KUKA KRL program: EPS_2_25716_MHCR06_A_20250905053017.src

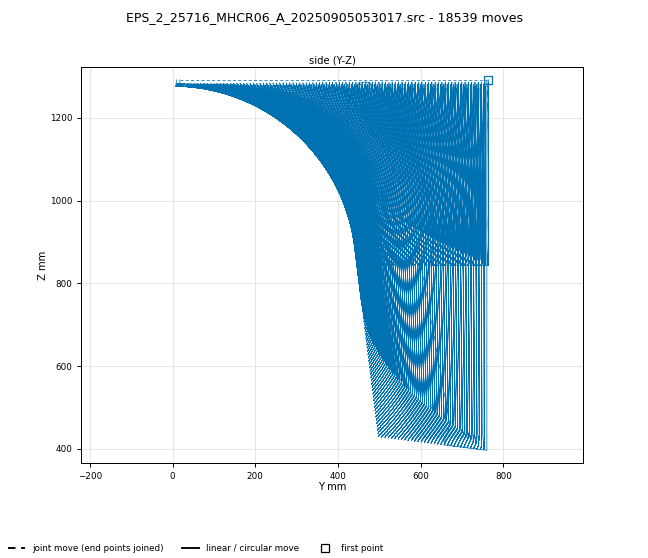
[picture p0: tool path of EPS_2_25716_MHCR06_A_20250905053017.src, 18539 of 18541 moves have a stored position in this frame; points joined in program order, loops and branches not executed]
&ACCESS RVP
&REL 4
&COMMENT QRS 19112012
&PARAM EDITMASK = *
DEF PART()
EXT BAS (BAS_COMMAND :IN,REAL :IN )
INT I
BAS (#INITMOV,0 )

;KUKA QRS Post kuka4.cps  Date:22-06-2017 !

File_ID=2806

QRS_PRE_INIT()

;Init var - Until changes are made in qrs_pre_init
Outlet_Square_prg=0
Inlet_1_Square_prg=0
Inlet_2_Square_prg=0
Inlet_3_Square_prg=0
Inlet_4_Square_prg=0
Inlet_5_Square_prg=0

Outlet_1={X 0.000, Y 457.000, Z 863.000, B 0.000, E1 0.000 }
Inlet_1={X 0.000, Y 457.000, Z 853.000, B 0.000, E1 180.000 }
Outlet_1_type=838
Inlet_1_type=838
;QRS#1=Sidecore dimensions
;QRS#2=825-33" Concrete
;QRS#3=825-33" Concrete
;QRS#4=
;QRS#5=
;QRS#6=
;QRS#7=
;QRS#8=
;QRS#9=S306-46
;QRS#10=S306-46
;QRS#11=
;QRS#12=
;QRS#13=
;QRS#14=
;QRS#15=
;QRS#16=1524x152x1753 5,75'
;QRS#17=EPS Height
;QRS#18=1282
;QRS#19=*
;QRS#20= UPDATED VERSION 22-06-2017
;QRS#21=*
Outlet_Square=0650
Inlet_1_Square=0650
Inlet_2_Square=0
Inlet_3_Square=0
Inlet_4_Square=0
Inlet_5_Square=0
Mill_Square=1
Outlet_Square_Prg=267
Inlet_1_Square_prg=267

QRS_INIT()

$ADVANCE=5

; T1
PTP {E1 176.612,E2 176.612}
PTP {X 0,Y 763.425,A -85,B 0,C 180,E1 176.612,E2 176.612,E3 0,E4 0,E5 0,E6 0}
QRS_SPEED_INIT()
LIN {X 0,Y 763.425,Z 1292,A -85,B 0,C 180,E1 176.612,E2 176.612,E3 0,E4 0,E5 0,E6 0} C_VEL
LIN {X 0,Y 763.425,Z 846.06,A -85,B 0,C 180,E1 176.612,E2 176.612} C_VEL
LIN {X 0,Y 763.534,Z 844.06,A -85,B 0,C 180,E1 176.762,E2 176.762} C_VEL
LIN {X 0,Y 763.871,Z 844.06,A -85,B 0,C 180,E1 177.187,E2 177.187} C_VEL
LIN {X 0,Y 763.823,Z 844.06,A -85,B 0,C 180,E1 184.692,E2 184.692} C_VEL
LIN {X 0,Y 763.818,Z 844.06,A -85,B 0,C 180,E1 192.28,E2 192.28} C_VEL
LIN {X 0,Y 763.836,Z 844.06,A -85,B 0,C 180,E1 200.095,E2 200.095} C_VEL
LIN {X 0,Y 763.785,Z 844.06,A -85,B 0,C 180,E1 208.327,E2 208.327} C_VEL
LIN {X 0,Y 762.377,Z 844.06,A -85,B 0,C 180,E1 210.541,E2 210.541} C_VEL
LIN {X 0,Y 762.698,Z 844.06,A -85,B 0,C 180,E1 214.994,E2 214.994} C_VEL
LIN {X 0,Y 763.696,Z 844.06,A -85,B 0,C 180,E1 216.695,E2 216.695} C_VEL
LIN {X 0,Y 763.424,Z 844.06,A -85,B 0,C 180,E1 224.741,E2 224.741} C_VEL
LIN {X 0,Y 763.668,Z 844.06,A -85,B 0,C 180,E1 225.277,E2 225.277} C_VEL
LIN {X 0,Y 763.811,Z 844.06,A -85,B 0,C 180,E1 233.406,E2 233.406} C_VEL
LIN {X 0,Y 763.414,Z 844.06,A -85,B 0,C 180,E1 233.624,E2 233.624} C_VEL
LIN {X 0,Y 763.044,Z 844.06,A -85,B 0,C 180,E1 233.668,E2 233.668} C_VEL
LIN {X 0,Y 762.773,Z 846.033,A -85,B 0,C 180,E1 233.717,E2 233.717} C_VEL
LIN {X 0,Y 763.464,Z 884.803,A -85,B 0,C 180,E1 234.197,E2 234.197} C_VEL
LIN {X 0,Y 763.74,Z 906.668,A -85,B 0,C 180,E1 234.483,E2 234.483} C_VEL
LIN {X 0,Y 763.751,Z 923.257,A -85,B 0,C 180,E1 234.748,E2 234.748} C_VEL
LIN {X 0,Y 763.617,Z 939.256,A -85,B 0,C 180,E1 235.054,E2 235.054} C_VEL
LIN {X 0,Y 763.249,Z 953.724,A -85,B 0,C 180,E1 235.362,E2 235.362} C_VEL
LIN {X 0,Y 763.625,Z 971.393,A -85,B 0,C 180,E1 235.846,E2 235.846} C_VEL
LIN {X 0,Y 763.699,Z 993.904,A -85,B 0,C 180,E1 236.542,E2 236.542} C_VEL
LIN {X 0,Y 763.605,Z 1014.167,A -85,B 0,C 180,E1 237.262,E2 237.262} C_VEL
LIN {X 0,Y 763.443,Z 1025.893,A -85,B 0,C 180,E1 237.721,E2 237.721} C_VEL
LIN {X 0,Y 763.576,Z 1034.178,A -85,B 0,C 180,E1 238.073,E2 238.073} C_VEL
LIN {X 0,Y 763.564,Z 1050.299,A -85,B 0,C 180,E1 238.794,E2 238.794} C_VEL
LIN {X 0,Y 763.558,Z 1067.921,A -85,B 0,C 180,E1 239.665,E2 239.665} C_VEL
LIN {X 0,Y 763.648,Z 1085.413,A -85,B 0,C 180,E1 240.62,E2 240.62} C_VEL
LIN {X 0,Y 763.58,Z 1101.247,A -85,B 0,C 180,E1 241.554,E2 241.554} C_VEL
LIN {X 0,Y 763.331,Z 1117.353,A -85,B 0,C 180,E1 242.582,E2 242.582} C_VEL
LIN {X 0,Y 763.287,Z 1132.396,A -85,B 0,C 180,E1 243.633,E2 243.633} C_VEL
LIN {X 0,Y 763.586,Z 1147.922,A -85,B 0,C 180,E1 244.824,E2 244.824} C_VEL
LIN {X 0,Y 763.68,Z 1158.714,A -85,B 0,C 180,E1 245.705,E2 245.705} C_VEL
LIN {X 0,Y 763.241,Z 1173.502,A -85,B 0,C 180,E1 246.987,E2 246.987} C_VEL
LIN {X 0,Y 763.107,Z 1186.863,A -85,B 0,C 180,E1 248.263,E2 248.263} C_VEL
LIN {X 0,Y 763.439,Z 1198.638,A -85,B 0,C 180,E1 249.493,E2 249.493} C_VEL
LIN {X 0,Y 763.75,Z 1205.883,A -85,B 0,C 180,E1 250.316,E2 250.316} C_VEL
LIN {X 0,Y 763.554,Z 1210.764,A -85,B 0,C 180,E1 250.869,E2 250.869} C_VEL
LIN {X 0,Y 762.975,Z 1220.993,A -85,B 0,C 180,E1 252.113,E2 252.113} C_VEL
LIN {X 0,Y 762.874,Z 1231.824,A -85,B 0,C 180,E1 253.584,E2 253.584} C_VEL
LIN {X 0,Y 763.518,Z 1241.781,A -85,B 0,C 180,E1 255.105,E2 255.105} C_VEL
LIN {X 0,Y 763.855,Z 1245.871,A -85,B 0,C 180,E1 255.793,E2 255.793} C_VEL
LIN {X 0,Y 763.464,Z 1249.702,A -85,B 0,C 180,E1 256.43,E2 256.43} C_VEL
LIN {X 0,Y 762.698,Z 1257.74,A -85,B 0,C 180,E1 257.94,E2 257.94} C_VEL
LIN {X 0,Y 762.694,Z 1264.404,A -85,B 0,C 180,E1 259.376,E2 259.376} C_VEL
LIN {X 0,Y 763.587,Z 1270.959,A -85,B 0,C 180,E1 261.054,E2 261.054} C_VEL
LIN {X 0,Y 763.866,Z 1272.551,A -85,B 0,C 180,E1 261.531,E2 261.531} C_VEL
LIN {X 0,Y 763.257,Z 1275.707,A -85,B 0,C 180,E1 262.472,E2 262.472} C_VEL
LIN {X 0,Y 762.641,Z 1279.586,A -85,B 0,C 180,E1 263.884,E2 263.884} C_VEL
LIN {X 0,Y 762.788,Z 1282.608,A -85,B 0,C 180,E1 265.299,E2 265.299} C_VEL
LIN {X 0,Y 763.582,Z 1284.794,A -85,B 0,C 180,E1 266.707,E2 266.707} C_VEL
LIN {X 0,Y 763.885,Z 1285.327,A -85,B 0,C 180,E1 267.185,E2 267.185} C_VEL
LIN {X 0,Y 762.666,Z 1286.718,A -85,B 0,C 180,E1 269.059,E2 269.059} C_VEL
LIN {X 0,Y 762.487,Z 1286.723,A -85,B 0,C 180,E1 270.937,E2 270.937} C_VEL
LIN {X 0,Y 763.544,Z 1285.349,A -85,B 0,C 180,E1 272.812,E2 272.812} C_VEL
LIN {X 0,Y 763.669,Z 1284.386,A -85,B 0,C 180,E1 273.591,E2 273.591} C_VEL
LIN {X 0,Y 763.006,Z 1282.612,A -85,B 0,C 180,E1 274.695,E2 274.695} C_VEL
LIN {X 0,Y 762.597,Z 1279.596,A -85,B 0,C 180,E1 276.112,E2 276.112} C_VEL
LIN {X 0,Y 762.981,Z 1275.722,A -85,B 0,C 180,E1 277.527,E2 277.527} C_VEL
LIN {X 0,Y 763.831,Z 1270.969,A -85,B 0,C 180,E1 278.939,E2 278.939} C_VEL
LIN {X 0,Y 763.296,Z 1267.291,A -85,B 0,C 180,E1 279.896,E2 279.896} C_VEL
LIN {X 0,Y 762.816,Z 1263.345,A -85,B 0,C 180,E1 280.857,E2 280.857} C_VEL
LIN {X 0,Y 762.703,Z 1256.562,A -85,B 0,C 180,E1 282.296,E2 282.296} C_VEL
LIN {X 0,Y 763.232,Z 1249.725,A -85,B 0,C 180,E1 283.57,E2 283.57} C_VEL
LIN {X 0,Y 763.817,Z 1243.189,A -85,B 0,C 180,E1 284.654,E2 284.654} C_VEL
LIN {X 0,Y 763.572,Z 1240.469,A -85,B 0,C 180,E1 285.11,E2 285.11} C_VEL
LIN {X 0,Y 762.935,Z 1230.124,A -85,B 0,C 180,E1 286.655,E2 286.655} C_VEL
LIN {X 0,Y 762.935,Z 1221.027,A -85,B 0,C 180,E1 287.883,E2 287.883} C_VEL
LIN {X 0,Y 763.482,Z 1209.87,A -85,B 0,C 180,E1 289.243,E2 289.243} C_VEL
LIN {X 0,Y 763.749,Z 1204.145,A -85,B 0,C 180,E1 289.879,E2 289.879} C_VEL
LIN {X 0,Y 763.45,Z 1196.64,A -85,B 0,C 180,E1 290.718,E2 290.718} C_VEL
LIN {X 0,Y 763.048,Z 1184.242,A -85,B 0,C 180,E1 291.997,E2 291.997} C_VEL
LIN {X 0,Y 763.138,Z 1172.143,A -85,B 0,C 180,E1 293.139,E2 293.139} C_VEL
LIN {X 0,Y 763.585,Z 1158.001,A -85,B 0,C 180,E1 294.356,E2 294.356} C_VEL
LIN {X 0,Y 763.639,Z 1146.811,A -85,B 0,C 180,E1 295.265,E2 295.265} C_VEL
LIN {X 0,Y 763.318,Z 1130.65,A -85,B 0,C 180,E1 296.492,E2 296.492} C_VEL
LIN {X 0,Y 763.302,Z 1114.416,A -85,B 0,C 180,E1 297.612,E2 297.612} C_VEL
LIN {X 0,Y 763.543,Z 1098.417,A -85,B 0,C 180,E1 298.618,E2 298.618} C_VEL
LIN {X 0,Y 763.622,Z 1082.558,A -85,B 0,C 180,E1 299.543,E2 299.543} C_VEL
LIN {X 0,Y 763.573,Z 1064.988,A -85,B 0,C 180,E1 300.484,E2 300.484} C_VEL
LIN {X 0,Y 763.534,Z 1047.236,A -85,B 0,C 180,E1 301.35,E2 301.35} C_VEL
LIN {X 0,Y 763.593,Z 1029.838,A -85,B 0,C 180,E1 302.115,E2 302.115} C_VEL
LIN {X 0,Y 763.413,Z 1015.501,A -85,B 0,C 180,E1 302.694,E2 302.694} C_VEL
LIN {X 0,Y 763.608,Z 1006.295,A -85,B 0,C 180,E1 303.025,E2 303.025} C_VEL
LIN {X 0,Y 763.703,Z 991.031,A -85,B 0,C 180,E1 303.552,E2 303.552} C_VEL
LIN {X 0,Y 763.676,Z 970.59,A -85,B 0,C 180,E1 304.173,E2 304.173} C_VEL
LIN {X 0,Y 763.496,Z 952.918,A -85,B 0,C 180,E1 304.645,E2 304.645} C_VEL
LIN {X 0,Y 763.248,Z 942.803,A -85,B 0,C 180,E1 304.891,E2 304.891} C_VEL
LIN {X 0,Y 763.633,Z 926.104,A -85,B 0,C 180,E1 305.206,E2 305.206} C_VEL
LIN {X 0,Y 763.708,Z 908.879,A -85,B 0,C 180,E1 305.487,E2 305.487} C_VEL
LIN {X 0,Y 763.624,Z 893.145,A -85,B 0,C 180,E1 305.699,E2 305.699} C_VEL
LIN {X 0,Y 762.84,Z 848.075,A -85,B 0,C 180,E1 306.256,E2 306.256} C_VEL
LIN {X 0,Y 763.386,Z 844.06,A -85,B 0,C 180,E1 306.373,E2 306.373} C_VEL
LIN {X 0,Y 763.822,Z 844.06,A -85,B 0,C 180,E1 306.471,E2 306.471} C_VEL
LIN {X 0,Y 763.69,Z 844.06,A -85,B 0,C 180,E1 312.133,E2 312.133} C_VEL
LIN {X 0,Y 763.519,Z 844.06,A -85,B 0,C 180,E1 312.562,E2 312.562} C_VEL
LIN {X 0,Y 763.784,Z 844.06,A -85,B 0,C 180,E1 320.259,E2 320.259} C_VEL
LIN {X 0,Y 763.636,Z 844.06,A -85,B 0,C 180,E1 326.569,E2 326.569} C_VEL
LIN {X 0,Y 763.395,Z 844.06,A -85,B 0,C 180,E1 327.301,E2 327.301} C_VEL
LIN {X 0,Y 763.767,Z 844.06,A -85,B 0,C 180,E1 333.782,E2 333.782} C_VEL
LIN {X 0,Y 763.774,Z 844.06,A -85,B 0,C 180,E1 341.888,E2 341.888} C_VEL
LIN {X 0,Y 763.762,Z 844.06,A -85,B 0,C 180,E1 349.631,E2 349.631} C_VEL
LIN {X 0,Y 763.87,Z 844.06,A -85,B 0,C 180,E1 357.187,E2 357.187} C_VEL
LIN {X 0,Y 763.811,Z 844.06,A -85,B 0,C 180,E1 364.692,E2 364.692} C_VEL
LIN {X 0,Y 763.783,Z 844.06,A -85,B 0,C 180,E1 372.281,E2 372.281} C_VEL
LIN {X 0,Y 763.826,Z 844.06,A -85,B 0,C 180,E1 380.095,E2 380.095} C_VEL
LIN {X 0,Y 763.817,Z 844.06,A -85,B 0,C 180,E1 388.325,E2 388.325} C_VEL
LIN {X 0,Y 762.037,Z 844.06,A -85,B 0,C 180,E1 393.248,E2 393.248} C_VEL
LIN {X 0,Y 762.694,Z 844.06,A -85,B 0,C 180,E1 394.994,E2 394.994} C_VEL
LIN {X 0,Y 763.695,Z 844.06,A -85,B 0,C 180,E1 396.702,E2 396.702} C_VEL
LIN {X 0,Y 763.462,Z 844.06,A -85,B 0,C 180,E1 404.738,E2 404.738} C_VEL
LIN {X 0,Y 763.718,Z 844.06,A -85,B 0,C 180,E1 405.287,E2 405.287} C_VEL
LIN {X 0,Y 763.716,Z 844.06,A -85,B 0,C 180,E1 413.316,E2 413.316} C_VEL
LIN {X 0,Y 763.638,Z 844.06,A -85,B 0,C 180,E1 413.584,E2 413.584} C_VEL
LIN {X 0,Y 762.291,Z 846.452,A -85,B 0,C 180,E1 413.765,E2 413.765} C_VEL
LIN {X 0,Y 763.273,Z 877.101,A -85,B 0,C 180,E1 414.168,E2 414.168} C_VEL
LIN {X 0,Y 763.588,Z 897.131,A -85,B 0,C 180,E1 414.436,E2 414.436} C_VEL
LIN {X 0,Y 763.619,Z 912.565,A -85,B 0,C 180,E1 414.683,E2 414.683} C_VEL
LIN {X 0,Y 763.39,Z 929.413,A -85,B 0,C 180,E1 415,E2 415} C_VEL
LIN {X 0,Y 763.232,Z 936.778,A -85,B 0,C 180,E1 415.154,E2 415.154} C_VEL
LIN {X 0,Y 763.582,Z 953.603,A -85,B 0,C 180,E1 415.585,E2 415.585} C_VEL
LIN {X 0,Y 763.631,Z 965.787,A -85,B 0,C 180,E1 415.931,E2 415.931} C_VEL
LIN {X 0,Y 763.567,Z 984.677,A -85,B 0,C 180,E1 416.518,E2 416.518} C_VEL
LIN {X 0,Y 763.383,Z 997.385,A -85,B 0,C 180,E1 416.957,E2 416.957} C_VEL
LIN {X 0,Y 763.555,Z 1005.386,A -85,B 0,C 180,E1 417.264,E2 417.264} C_VEL
LIN {X 0,Y 763.596,Z 1022.442,A -85,B 0,C 180,E1 417.952,E2 417.952} C_VEL
LIN {X 0,Y 763.616,Z 1040.545,A -85,B 0,C 180,E1 418.764,E2 418.764} C_VEL
LIN {X 0,Y 763.625,Z 1058.696,A -85,B 0,C 180,E1 419.665,E2 419.665} C_VEL
LIN {X 0,Y 763.566,Z 1074.602,A -85,B 0,C 180,E1 420.523,E2 420.523} C_VEL
LIN {X 0,Y 763.386,Z 1091.268,A -85,B 0,C 180,E1 421.502,E2 421.502} C_VEL
LIN {X 0,Y 763.398,Z 1108.066,A -85,B 0,C 180,E1 422.59,E2 422.59} C_VEL
LIN {X 0,Y 763.623,Z 1123.055,A -85,B 0,C 180,E1 423.65,E2 423.65} C_VEL
LIN {X 0,Y 763.542,Z 1136.934,A -85,B 0,C 180,E1 424.697,E2 424.697} C_VEL
LIN {X 0,Y 763.195,Z 1151.007,A -85,B 0,C 180,E1 425.838,E2 425.838} C_VEL
LIN {X 0,Y 763.158,Z 1164.022,A -85,B 0,C 180,E1 426.989,E2 426.989} C_VEL
LIN {X 0,Y 763.569,Z 1177.101,A -85,B 0,C 180,E1 428.256,E2 428.256} C_VEL
LIN {X 0,Y 763.758,Z 1183.715,A -85,B 0,C 180,E1 428.945,E2 428.945} C_VEL
LIN {X 0,Y 763.477,Z 1190.192,A -85,B 0,C 180,E1 429.624,E2 429.624} C_VEL
LIN {X 0,Y 762.964,Z 1201.113,A -85,B 0,C 180,E1 430.851,E2 430.851} C_VEL
LIN {X 0,Y 762.921,Z 1211.36,A -85,B 0,C 180,E1 432.116,E2 432.116} C_VEL
LIN {X 0,Y 763.535,Z 1222.154,A -85,B 0,C 180,E1 433.603,E2 433.603} C_VEL
LIN {X 0,Y 763.785,Z 1225.597,A -85,B 0,C 180,E1 434.123,E2 434.123} C_VEL
LIN {X 0,Y 763.432,Z 1230.981,A -85,B 0,C 180,E1 434.925,E2 434.925} C_VEL
LIN {X 0,Y 762.734,Z 1239.964,A -85,B 0,C 180,E1 436.421,E2 436.421} C_VEL
LIN {X 0,Y 762.83,Z 1247.97,A -85,B 0,C 180,E1 437.946,E2 437.946} C_VEL
LIN {X 0,Y 763.595,Z 1254.602,A -85,B 0,C 180,E1 439.393,E2 439.393} C_VEL
LIN {X 0,Y 763.746,Z 1255.557,A -85,B 0,C 180,E1 439.633,E2 439.633} C_VEL
LIN {X 0,Y 763.715,Z 1257.47,A -85,B 0,C 180,E1 440.109,E2 440.109} C_VEL
LIN {X 0,Y 763.137,Z 1261.129,A -85,B 0,C 180,E1 441.053,E2 441.053} C_VEL
LIN {X 0,Y 762.635,Z 1265.853,A -85,B 0,C 180,E1 442.47,E2 442.47} C_VEL
LIN {X 0,Y 762.909,Z 1269.7,A -85,B 0,C 180,E1 443.89,E2 443.89} C_VEL
LIN {X 0,Y 763.739,Z 1272.676,A -85,B 0,C 180,E1 445.309,E2 445.309} C_VEL
LIN {X 0,Y 763.388,Z 1274.244,A -85,B 0,C 180,E1 446.248,E2 446.248} C_VEL
LIN {X 0,Y 762.851,Z 1275.415,A -85,B 0,C 180,E1 447.185,E2 447.185} C_VEL
LIN {X 0,Y 762.523,Z 1276.623,A -85,B 0,C 180,E1 448.683,E2 448.683} C_VEL
LIN {X 0,Y 762.622,Z 1276.734,A -85,B 0,C 180,E1 449.063,E2 449.063} C_VEL
LIN {X 0,Y 763.558,Z 1276.671,A -85,B 0,C 180,E1 450.94,E2 450.94} C_VEL
LIN {X 0,Y 763.081,Z 1275.324,A -85,B 0,C 180,E1 452.818,E2 452.818} C_VEL
LIN {X 0,Y 762.778,Z 1274.133,A -85,B 0,C 180,E1 453.76,E2 453.76} C_VEL
LIN {X 0,Y 762.828,Z 1272.519,A -85,B 0,C 180,E1 454.7,E2 454.7} C_VEL
LIN {X 0,Y 763.445,Z 1269.457,A -85,B 0,C 180,E1 456.11,E2 456.11} C_VEL
LIN {X 0,Y 763.721,Z 1268.228,A -85,B 0,C 180,E1 456.579,E2 456.579} C_VEL
LIN {X 0,Y 763.733,Z 1266.935,A -85,B 0,C 180,E1 457.051,E2 457.051} C_VEL
LIN {X 0,Y 763.169,Z 1264.012,A -85,B 0,C 180,E1 458.003,E2 458.003} C_VEL
LIN {X 0,Y 762.74,Z 1260.812,A -85,B 0,C 180,E1 458.956,E2 458.956} C_VEL
LIN {X 0,Y 762.783,Z 1254.219,A -85,B 0,C 180,E1 460.623,E2 460.623} C_VEL
LIN {X 0,Y 763.718,Z 1246.298,A -85,B 0,C 180,E1 462.284,E2 462.284} C_VEL
LIN {X 0,Y 763.866,Z 1245.018,A -85,B 0,C 180,E1 462.521,E2 462.521} C_VEL
LIN {X 0,Y 763.236,Z 1238.998,A -85,B 0,C 180,E1 463.655,E2 463.655} C_VEL
LIN {X 0,Y 762.746,Z 1231.289,A -85,B 0,C 180,E1 464.948,E2 464.948} C_VEL
LIN {X 0,Y 762.932,Z 1221.523,A -85,B 0,C 180,E1 466.415,E2 466.415} C_VEL
LIN {X 0,Y 763.743,Z 1209.644,A -85,B 0,C 180,E1 467.991,E2 467.991} C_VEL
LIN {X 0,Y 763.596,Z 1204.366,A -85,B 0,C 180,E1 468.642,E2 468.642} C_VEL
LIN {X 0,Y 763.241,Z 1198.049,A -85,B 0,C 180,E1 469.41,E2 469.41} C_VEL
LIN {X 0,Y 762.917,Z 1187.203,A -85,B 0,C 180,E1 470.63,E2 470.63} C_VEL
LIN {X 0,Y 763.125,Z 1175.234,A -85,B 0,C 180,E1 471.855,E2 471.855} C_VEL
LIN {X 0,Y 763.677,Z 1161.576,A -85,B 0,C 180,E1 473.127,E2 473.127} C_VEL
LIN {X 0,Y 763.635,Z 1152.845,A -85,B 0,C 180,E1 473.895,E2 473.895} C_VEL
LIN {X 0,Y 763.447,Z 1146.602,A -85,B 0,C 180,E1 474.429,E2 474.429} C_VEL
LIN {X 0,Y 763.194,Z 1135.008,A -85,B 0,C 180,E1 475.376,E2 475.376} C_VEL
LIN {X 0,Y 763.25,Z 1119.932,A -85,B 0,C 180,E1 476.5,E2 476.5} C_VEL
LIN {X 0,Y 763.557,Z 1104.671,A -85,B 0,C 180,E1 477.541,E2 477.541} C_VEL
LIN {X 0,Y 763.635,Z 1089.28,A -85,B 0,C 180,E1 478.519,E2 478.519} C_VEL
LIN {X 0,Y 763.475,Z 1072.12,A -85,B 0,C 180,E1 479.528,E2 479.528} C_VEL
LIN {X 0,Y 763.463,Z 1055.627,A -85,B 0,C 180,E1 480.413,E2 480.413} C_VEL
LIN {X 0,Y 763.569,Z 1037.373,A -85,B 0,C 180,E1 481.297,E2 481.297} C_VEL
LIN {X 0,Y 763.485,Z 1023.615,A -85,B 0,C 180,E1 481.911,E2 481.911} C_VEL
LIN {X 0,Y 763.635,Z 1013.736,A -85,B 0,C 180,E1 482.31,E2 482.31} C_VEL
LIN {X 0,Y 763.68,Z 1000.1,A -85,B 0,C 180,E1 482.843,E2 482.843} C_VEL
LIN {X 0,Y 763.672,Z 981.403,A -85,B 0,C 180,E1 483.497,E2 483.497} C_VEL
LIN {X 0,Y 763.529,Z 959.922,A -85,B 0,C 180,E1 484.154,E2 484.154} C_VEL
LIN {X 0,Y 763.267,Z 949.422,A -85,B 0,C 180,E1 484.448,E2 484.448} C_VEL
LIN {X 0,Y 763.638,Z 933.768,A -85,B 0,C 180,E1 484.804,E2 484.804} C_VEL
LIN {X 0,Y 763.72,Z 917.765,A -85,B 0,C 180,E1 485.125,E2 485.125} C_VEL
LIN {X 0,Y 763.655,Z 901.543,A -85,B 0,C 180,E1 485.406,E2 485.406} C_VEL
LIN {X 0,Y 763.323,Z 882.8,A -85,B 0,C 180,E1 485.675,E2 485.675} C_VEL
LIN {X 0,Y 762.34,Z 860.304,A -85,B 0,C 180,E1 485.984,E2 485.984} C_VEL
LIN {X 0,Y 761.284,Z 844.06,A -85,B 0,C 180,E1 486.23,E2 486.23} C_VEL
LIN {X 0,Y 761.82,Z 844.06,A -85,B 0,C 180,E1 486.25,E2 486.25} C_VEL
LIN {X 0,Y 762.919,Z 844.06,A -85,B 0,C 180,E1 486.319,E2 486.319} C_VEL
LIN {X 0,Y 763.876,Z 844.06,A -85,B 0,C 180,E1 486.504,E2 486.504} C_VEL
LIN {X 0,Y 763.739,Z 844.06,A -85,B 0,C 180,E1 494.718,E2 494.718} C_VEL
LIN {X 0,Y 763.524,Z 844.06,A -85,B 0,C 180,E1 495.267,E2 495.267} C_VEL
LIN {X 0,Y 762.402,Z 844.06,A -85,B 0,C 180,E1 500.391,E2 500.391} C_VEL
LIN {X 0,Y 763.754,Z 844.06,A -85,B 0,C 180,E1 502.741,E2 502.741} C_VEL
LIN {X 0,Y 763.659,Z 844.06,A -85,B 0,C 180,E1 510.15,E2 510.15} C_VEL
LIN {X 0,Y 762.952,Z 844.06,A -85,B 0,C 180,E1 511.64,E2 511.64} C_VEL
LIN {X 0,Y 763.815,Z 844.06,A -85,B 0,C 180,E1 517.895,E2 517.895} C_VEL
LIN {X 0,Y 763.503,Z 844.06,A -85,B 0,C 180,E1 524.952,E2 524.952} C_VEL
LIN {X 0,Y 763.698,Z 844.06,A -85,B 0,C 180,E1 525.791,E2 525.791} C_VEL
LIN {X 0,Y 763.864,Z 844.06,A -85,B 0,C 180,E1 529.632,E2 529.632} C_VEL
LIN {X 0,Y 763.534,Z 844.06,A -85,B 0,C 180,E1 536.762,E2 536.762} C_VEL
LIN {X 0,Y 754.507,Z 844.06,A -85,B 0,C 180,E1 539.36,E2 539.36} C_VEL
LIN {X 0,Y 754.69,Z 844.06,A -85,B 0,C 180,E1 546.329,E2 546.329} C_VEL
LIN {X 0,Y 755.007,Z 844.06,A -85,B 0,C 180,E1 553.341,E2 553.341} C_VEL
LIN {X 0,Y 755.088,Z 844.06,A -85,B 0,C 180,E1 560.946,E2 560.946} C_VEL
LIN {X 0,Y 754.916,Z 844.06,A -85,B 0,C 180,E1 569.473,E2 569.473} C_VEL
LIN {X 0,Y 754.765,Z 844.06,A -85,B 0,C 180,E1 577.785,E2 577.785} C_VEL
LIN {X 0,Y 754.965,Z 844.06,A -85,B 0,C 180,E1 586.13,E2 586.13} C_VEL
LIN {X 0,Y 755.974,Z 846.019,A -85,B 0,C 180,E1 593.338,E2 593.338} C_VEL
LIN {X 0,Y 756.776,Z 949.003,A -85,B 0,C 180,E1 594.911,E2 594.911} C_VEL
LIN {X 0,Y 756.504,Z 1025.149,A -85,B 0,C 180,E1 597.359,E2 597.359} C_VEL
LIN {X 0,Y 756.265,Z 1095.442,A -85,B 0,C 180,E1 600.903,E2 600.903} C_VEL
LIN {X 0,Y 756.017,Z 1158.226,A -85,B 0,C 180,E1 605.403,E2 605.403} C_VEL
LIN {X 0,Y 755.77,Z 1210.774,A -85,B 0,C 180,E1 610.665,E2 610.665} C_VEL
LIN {X 0,Y 755.535,Z 1250.09,A -85,B 0,C 180,E1 616.358,E2 616.358} C_VEL
LIN {X 0,Y 755.248,Z 1276.023,A -85,B 0,C 180,E1 622.5,E2 622.5} C_VEL
LIN {X 0,Y 755.095,Z 1286.378,A -85,B 0,C 180,E1 628.274,E2 628.274} C_VEL
LIN {X 0,Y 755.382,Z 1283.831,A -85,B 0,C 180,E1 634.029,E2 634.029} C_VEL
LIN {X 0,Y 755.203,Z 1266.829,A -85,B 0,C 180,E1 640.12,E2 640.12} C_VEL
LIN {X 0,Y 755.335,Z 1237.502,A -85,B 0,C 180,E1 645.727,E2 645.727} C_VEL
LIN {X 0,Y 755.493,Z 1193.664,A -85,B 0,C 180,E1 651.257,E2 651.257} C_VEL
LIN {X 0,Y 755.86,Z 1137.282,A -85,B 0,C 180,E1 656.273,E2 656.273} C_VEL
LIN {X 0,Y 756.384,Z 1070.763,A -85,B 0,C 180,E1 660.498,E2 660.498} C_VEL
LIN {X 0,Y 756.832,Z 999.111,A -85,B 0,C 180,E1 663.616,E2 663.616} C_VEL
LIN {X 0,Y 757.076,Z 926.301,A -85,B 0,C 180,E1 665.553,E2 665.553} C_VEL
LIN {X 0,Y 755.648,Z 844.06,A -85,B 0,C 180,E1 666.742,E2 666.742} C_VEL
LIN {X 0,Y 754.602,Z 844.06,A -85,B 0,C 180,E1 673.896,E2 673.896} C_VEL
LIN {X 0,Y 755.415,Z 844.06,A -85,B 0,C 180,E1 680.783,E2 680.783} C_VEL
LIN {X 0,Y 755.055,Z 844.06,A -85,B 0,C 180,E1 687.852,E2 687.852} C_VEL
LIN {X 0,Y 755.211,Z 844.06,A -85,B 0,C 180,E1 694.434,E2 694.434} C_VEL
LIN {X 0,Y 754.86,Z 844.06,A -85,B 0,C 180,E1 703.078,E2 703.078} C_VEL
LIN {X 0,Y 755.31,Z 844.06,A -85,B 0,C 180,E1 710.189,E2 710.189} C_VEL
LIN {X 0,Y 755.035,Z 844.06,A -85,B 0,C 180,E1 718.292,E2 718.292} C_VEL
LIN {X 0,Y 754.837,Z 844.06,A -85,B 0,C 180,E1 726.012,E2 726.012} C_VEL
LIN {X 0,Y 754.927,Z 844.06,A -85,B 0,C 180,E1 733.381,E2 733.381} C_VEL
LIN {X 0,Y 755.092,Z 844.06,A -85,B 0,C 180,E1 740.947,E2 740.947} C_VEL
LIN {X 0,Y 754.864,Z 844.06,A -85,B 0,C 180,E1 749.518,E2 749.518} C_VEL
LIN {X 0,Y 754.768,Z 844.06,A -85,B 0,C 180,E1 757.832,E2 757.832} C_VEL
LIN {X 0,Y 755.021,Z 844.06,A -85,B 0,C 180,E1 766.135,E2 766.135} C_VEL
LIN {X 0,Y 755.758,Z 844.957,A -85,B 0,C 180,E1 773.384,E2 773.384} C_VEL
LIN {X 0,Y 756.697,Z 941.68,A -85,B 0,C 180,E1 774.924,E2 774.924} C_VEL
LIN {X 0,Y 756.626,Z 1017.331,A -85,B 0,C 180,E1 777.407,E2 777.407} C_VEL
LIN {X 0,Y 756.084,Z 1088.961,A -85,B 0,C 180,E1 781.06,E2 781.06} C_VEL
LIN {X 0,Y 755.615,Z 1150.628,A -85,B 0,C 180,E1 785.547,E2 785.547} C_VEL
LIN {X 0,Y 755.163,Z 1201.136,A -85,B 0,C 180,E1 790.649,E2 790.649} C_VEL
LIN {X 0,Y 755.024,Z 1236.932,A -85,B 0,C 180,E1 795.756,E2 795.756} C_VEL
LIN {X 0,Y 755.321,Z 1260.454,A -85,B 0,C 180,E1 800.757,E2 800.757} C_VEL
LIN {X 0,Y 755.469,Z 1273.905,A -85,B 0,C 180,E1 805.971,E2 805.971} C_VEL
LIN {X 0,Y 755.269,Z 1276.338,A -85,B 0,C 180,E1 811.726,E2 811.726} C_VEL
LIN {X 0,Y 755.445,Z 1265.894,A -85,B 0,C 180,E1 817.498,E2 817.498} C_VEL
LIN {X 0,Y 755.43,Z 1241.41,A -85,B 0,C 180,E1 823.348,E2 823.348} C_VEL
LIN {X 0,Y 755.57,Z 1202.857,A -85,B 0,C 180,E1 829.036,E2 829.036} C_VEL
LIN {X 0,Y 755.887,Z 1151.386,A -85,B 0,C 180,E1 834.286,E2 834.286} C_VEL
LIN {X 0,Y 756.272,Z 1088.823,A -85,B 0,C 180,E1 838.85,E2 838.85} C_VEL
LIN {X 0,Y 756.638,Z 1019.327,A -85,B 0,C 180,E1 842.422,E2 842.422} C_VEL
LIN {X 0,Y 756.797,Z 944.281,A -85,B 0,C 180,E1 844.917,E2 844.917} C_VEL
LIN {X 0,Y 755.099,Z 849.345,A -85,B 0,C 180,E1 846.512,E2 846.512} C_VEL
LIN {X 0,Y 755.653,Z 844.06,A -85,B 0,C 180,E1 846.66,E2 846.66} C_VEL
LIN {X 0,Y 754.933,Z 844.06,A -85,B 0,C 180,E1 856.084,E2 856.084} C_VEL
LIN {X 0,Y 755.077,Z 844.06,A -85,B 0,C 180,E1 863.629,E2 863.629} C_VEL
LIN {X 0,Y 754.878,Z 844.06,A -85,B 0,C 180,E1 871.797,E2 871.797} C_VEL
LIN {X 0,Y 754.777,Z 844.06,A -85,B 0,C 180,E1 879.387,E2 879.387} C_VEL
LIN {X 0,Y 755.412,Z 844.06,A -85,B 0,C 180,E1 886.822,E2 886.822} C_VEL
LIN {X 0,Y 754.234,Z 844.06,A -85,B 0,C 180,E1 893.63,E2 893.63} C_VEL
LIN {X 0,Y 755.082,Z 844.06,A -85,B 0,C 180,E1 898.254,E2 898.254} C_VEL
LIN {X 0,Y 754.507,Z 844.06,A -85,B 0,C 180,E1 899.36,E2 899.36} C_VEL
LIN {X 0,Y 746.363,Z 844.06,A -85,B 0,C 180,E1 901.991,E2 901.991} C_VEL
LIN {X 0,Y 746.244,Z 844.06,A -85,B 0,C 180,E1 907.574,E2 907.574} C_VEL
LIN {X 0,Y 746.903,Z 844.06,A -85,B 0,C 180,E1 913.488,E2 913.488} C_VEL
LIN {X 0,Y 747.2,Z 844.06,A -85,B 0,C 180,E1 920.792,E2 920.792} C_VEL
LIN {X 0,Y 747.444,Z 844.06,A -85,B 0,C 180,E1 928.466,E2 928.466} C_VEL
LIN {X 0,Y 747.225,Z 844.06,A -85,B 0,C 180,E1 936.769,E2 936.769} C_VEL
LIN {X 0,Y 746.97,Z 844.06,A -85,B 0,C 180,E1 946.108,E2 946.108} C_VEL
LIN {X 0,Y 747.497,Z 845.875,A -85,B 0,C 180,E1 952.851,E2 952.851} C_VEL
LIN {X 0,Y 750.115,Z 861.338,A -85,B 0,C 180,E1 953.184,E2 953.184} C_VEL
LIN {X 0,Y 750.091,Z 952.668,A -85,B 0,C 180,E1 954.638,E2 954.638} C_VEL
LIN {X 0,Y 749.533,Z 1028.886,A -85,B 0,C 180,E1 957.169,E2 957.169} C_VEL
LIN {X 0,Y 748.946,Z 1100.374,A -85,B 0,C 180,E1 960.889,E2 960.889} C_VEL
LIN {X 0,Y 748.331,Z 1162.953,A -85,B 0,C 180,E1 965.549,E2 965.549} C_VEL
LIN {X 0,Y 747.716,Z 1214.832,A -85,B 0,C 180,E1 970.959,E2 970.959} C_VEL
LIN {X 0,Y 747.444,Z 1251.648,A -85,B 0,C 180,E1 976.507,E2 976.507} C_VEL
LIN {X 0,Y 747.286,Z 1276.023,A -85,B 0,C 180,E1 982.42,E2 982.42} C_VEL
LIN {X 0,Y 747.099,Z 1286.379,A -85,B 0,C 180,E1 988.255,E2 988.255} C_VEL
LIN {X 0,Y 747.365,Z 1283.831,A -85,B 0,C 180,E1 994.073,E2 994.073} C_VEL
LIN {X 0,Y 747.219,Z 1267.121,A -85,B 0,C 180,E1 1000.155,E2 1000.155} C_VEL
LIN {X 0,Y 747.349,Z 1237.503,A -85,B 0,C 180,E1 1005.899,E2 1005.899} C_VEL
LIN {X 0,Y 747.663,Z 1193.888,A -85,B 0,C 180,E1 1011.467,E2 1011.467} C_VEL
LIN {X 0,Y 748.31,Z 1137.999,A -85,B 0,C 180,E1 1016.504,E2 1016.504} C_VEL
LIN {X 0,Y 749.207,Z 1071.667,A -85,B 0,C 180,E1 1020.772,E2 1020.772} C_VEL
LIN {X 0,Y 750.007,Z 1000.491,A -85,B 0,C 180,E1 1023.913,E2 1023.913} C_VEL
LIN {X 0,Y 750.53,Z 926.375,A -85,B 0,C 180,E1 1025.91,E2 1025.91} C_VEL
LIN {X 0,Y 748.238,Z 847.51,A -85,B 0,C 180,E1 1027.087,E2 1027.087} C_VEL
LIN {X 0,Y 747.316,Z 844.06,A -85,B 0,C 180,E1 1027.332,E2 1027.332} C_VEL
LIN {X 0,Y 746.614,Z 844.06,A -85,B 0,C 180,E1 1033.864,E2 1033.864} C_VEL
LIN {X 0,Y 746.91,Z 844.06,A -85,B 0,C 180,E1 1041.746,E2 1041.746} C_VEL
LIN {X 0,Y 746.627,Z 844.06,A -85,B 0,C 180,E1 1048.816,E2 1048.816} C_VEL
LIN {X 0,Y 746.544,Z 844.06,A -85,B 0,C 180,E1 1055.402,E2 1055.402} C_VEL
LIN {X 0,Y 746.984,Z 844.06,A -85,B 0,C 180,E1 1062.894,E2 1062.894} C_VEL
LIN {X 0,Y 747.291,Z 844.06,A -85,B 0,C 180,E1 1070.083,E2 1070.083} C_VEL
LIN {X 0,Y 747.039,Z 844.06,A -85,B 0,C 180,E1 1078.273,E2 1078.273} C_VEL
LIN {X 0,Y 747.359,Z 844.06,A -85,B 0,C 180,E1 1085.26,E2 1085.26} C_VEL
LIN {X 0,Y 746.83,Z 844.06,A -85,B 0,C 180,E1 1093.528,E2 1093.528} C_VEL
LIN {X 0,Y 747.18,Z 844.06,A -85,B 0,C 180,E1 1100.833,E2 1100.833} C_VEL
LIN {X 0,Y 747.461,Z 844.06,A -85,B 0,C 180,E1 1108.508,E2 1108.508} C_VEL
LIN {X 0,Y 747.245,Z 844.06,A -85,B 0,C 180,E1 1116.815,E2 1116.815} C_VEL
LIN {X 0,Y 746.991,Z 844.06,A -85,B 0,C 180,E1 1126.16,E2 1126.16} C_VEL
LIN {X 0,Y 747.582,Z 845.894,A -85,B 0,C 180,E1 1132.929,E2 1132.929} C_VEL
LIN {X 0,Y 750.583,Z 901.878,A -85,B 0,C 180,E1 1133.795,E2 1133.795} C_VEL
LIN {X 0,Y 750.12,Z 971.219,A -85,B 0,C 180,E1 1135.403,E2 1135.403} C_VEL
LIN {X 0,Y 749.451,Z 1042.609,A -85,B 0,C 180,E1 1138.21,E2 1138.21} C_VEL
LIN {X 0,Y 748.492,Z 1110.871,A -85,B 0,C 180,E1 1142.198,E2 1142.198} C_VEL
LIN {X 0,Y 747.779,Z 1170.456,A -85,B 0,C 180,E1 1147.116,E2 1147.116} C_VEL
LIN {X 0,Y 747.255,Z 1216.624,A -85,B 0,C 180,E1 1152.457,E2 1152.457} C_VEL
LIN {X 0,Y 746.845,Z 1247.991,A -85,B 0,C 180,E1 1157.689,E2 1157.689} C_VEL
LIN {X 0,Y 746.672,Z 1266.151,A -85,B 0,C 180,E1 1162.414,E2 1162.414} C_VEL
LIN {X 0,Y 746.907,Z 1275.395,A -85,B 0,C 180,E1 1167.09,E2 1167.09} C_VEL
LIN {X 0,Y 747.078,Z 1275.315,A -85,B 0,C 180,E1 1172.909,E2 1172.909} C_VEL
LIN {X 0,Y 747.138,Z 1264.04,A -85,B 0,C 180,E1 1178.169,E2 1178.169} C_VEL
LIN {X 0,Y 747.271,Z 1239.858,A -85,B 0,C 180,E1 1183.796,E2 1183.796} C_VEL
LIN {X 0,Y 747.559,Z 1200.42,A -85,B 0,C 180,E1 1189.556,E2 1189.556} C_VEL
LIN {X 0,Y 748.139,Z 1147.416,A -85,B 0,C 180,E1 1194.896,E2 1194.896} C_VEL
LIN {X 0,Y 748.922,Z 1084.248,A -85,B 0,C 180,E1 1199.437,E2 1199.437} C_VEL
LIN {X 0,Y 749.782,Z 1013.463,A -85,B 0,C 180,E1 1202.995,E2 1202.995} C_VEL
LIN {X 0,Y 750.338,Z 938.46,A -85,B 0,C 180,E1 1205.403,E2 1205.403} C_VEL
LIN {X 0,Y 747.382,Z 844.06,A -85,B 0,C 180,E1 1207.044,E2 1207.044} C_VEL
LIN {X 0,Y 746.904,Z 844.06,A -85,B 0,C 180,E1 1216.121,E2 1216.121} C_VEL
LIN {X 0,Y 747.169,Z 844.06,A -85,B 0,C 180,E1 1223.296,E2 1223.296} C_VEL
LIN {X 0,Y 746.745,Z 844.06,A -85,B 0,C 180,E1 1232.058,E2 1232.058} C_VEL
LIN {X 0,Y 746.919,Z 844.06,A -85,B 0,C 180,E1 1239.16,E2 1239.16} C_VEL
LIN {X 0,Y 747.385,Z 844.06,A -85,B 0,C 180,E1 1247.675,E2 1247.675} C_VEL
LIN {X 0,Y 747.769,Z 844.06,A -85,B 0,C 180,E1 1257.074,E2 1257.074} C_VEL
LIN {X 0,Y 746.363,Z 844.06,A -85,B 0,C 180,E1 1261.991,E2 1261.991} C_VEL
LIN {X 0,Y 739.281,Z 844.06,A -85,B 0,C 180,E1 1264.672,E2 1264.672} C_VEL
LIN {X 0,Y 738.828,Z 844.06,A -85,B 0,C 180,E1 1273.639,E2 1273.639} C_VEL
LIN {X 0,Y 739.023,Z 844.06,A -85,B 0,C 180,E1 1281.033,E2 1281.033} C_VEL
LIN {X 0,Y 738.959,Z 844.06,A -85,B 0,C 180,E1 1289.283,E2 1289.283} C_VEL
LIN {X 0,Y 738.661,Z 844.06,A -85,B 0,C 180,E1 1297.773,E2 1297.773} C_VEL
LIN {X 0,Y 738.698,Z 844.06,A -85,B 0,C 180,E1 1306.548,E2 1306.548} C_VEL
LIN {X 0,Y 739.048,Z 845.552,A -85,B 0,C 180,E1 1312.349,E2 1312.349} C_VEL
LIN {X 0,Y 743.647,Z 858.977,A -85,B 0,C 180,E1 1312.782,E2 1312.782} C_VEL
LIN {X 0,Y 743.531,Z 952.122,A -85,B 0,C 180,E1 1314.265,E2 1314.265} C_VEL
LIN {X 0,Y 742.634,Z 1028.89,A -85,B 0,C 180,E1 1316.824,E2 1316.824} C_VEL
LIN {X 0,Y 741.636,Z 1100.467,A -85,B 0,C 180,E1 1320.58,E2 1320.58} C_VEL
LIN {X 0,Y 740.73,Z 1161.892,A -85,B 0,C 180,E1 1325.184,E2 1325.184} C_VEL
LIN {X 0,Y 740.045,Z 1213.229,A -85,B 0,C 180,E1 1330.55,E2 1330.55} C_VEL
LIN {X 0,Y 739.563,Z 1251.649,A -85,B 0,C 180,E1 1336.36,E2 1336.36} C_VEL
LIN {X 0,Y 739.343,Z 1276.023,A -85,B 0,C 180,E1 1342.338,E2 1342.338} C_VEL
LIN {X 0,Y 739.103,Z 1286.379,A -85,B 0,C 180,E1 1348.236,E2 1348.236} C_VEL
LIN {X 0,Y 739.33,Z 1283.831,A -85,B 0,C 180,E1 1354.117,E2 1354.117} C_VEL
LIN {X 0,Y 739.162,Z 1267.122,A -85,B 0,C 180,E1 1360.267,E2 1360.267} C_VEL
LIN {X 0,Y 739.369,Z 1237.505,A -85,B 0,C 180,E1 1366.075,E2 1366.075} C_VEL
LIN {X 0,Y 739.828,Z 1194.134,A -85,B 0,C 180,E1 1371.679,E2 1371.679} C_VEL
LIN {X 0,Y 740.74,Z 1137.446,A -85,B 0,C 180,E1 1376.839,E2 1376.839} C_VEL
LIN {X 0,Y 742.031,Z 1071.944,A -85,B 0,C 180,E1 1381.087,E2 1381.087} C_VEL
LIN {X 0,Y 743.196,Z 1000.333,A -85,B 0,C 180,E1 1384.273,E2 1384.273} C_VEL
LIN {X 0,Y 744.035,Z 926.39,A -85,B 0,C 180,E1 1386.272,E2 1386.272} C_VEL
LIN {X 0,Y 742.015,Z 850.415,A -85,B 0,C 180,E1 1387.416,E2 1387.416} C_VEL
LIN {X 0,Y 739.112,Z 844.06,A -85,B 0,C 180,E1 1387.826,E2 1387.826} C_VEL
LIN {X 0,Y 738.873,Z 844.06,A -85,B 0,C 180,E1 1393.439,E2 1393.439} C_VEL
LIN {X 0,Y 739.099,Z 844.06,A -85,B 0,C 180,E1 1401.267,E2 1401.267} C_VEL
LIN {X 0,Y 738.733,Z 844.06,A -85,B 0,C 180,E1 1408.445,E2 1408.445} C_VEL
LIN {X 0,Y 738.706,Z 844.06,A -85,B 0,C 180,E1 1415.124,E2 1415.124} C_VEL
LIN {X 0,Y 739.05,Z 844.06,A -85,B 0,C 180,E1 1422.704,E2 1422.704} C_VEL
LIN {X 0,Y 738.708,Z 844.06,A -85,B 0,C 180,E1 1431.159,E2 1431.159} C_VEL
LIN {X 0,Y 739.042,Z 844.06,A -85,B 0,C 180,E1 1438.255,E2 1438.255} C_VEL
LIN {X 0,Y 739.09,Z 844.06,A -85,B 0,C 180,E1 1445.635,E2 1445.635} C_VEL
LIN {X 0,Y 738.747,Z 844.06,A -85,B 0,C 180,E1 1453.679,E2 1453.679} C_VEL
LIN {X 0,Y 738.986,Z 844.06,A -85,B 0,C 180,E1 1461.075,E2 1461.075} C_VEL
LIN {X 0,Y 738.953,Z 844.06,A -85,B 0,C 180,E1 1469.283,E2 1469.283} C_VEL
LIN {X 0,Y 738.695,Z 844.06,A -85,B 0,C 180,E1 1477.777,E2 1477.777} C_VEL
LIN {X 0,Y 738.745,Z 844.06,A -85,B 0,C 180,E1 1486.551,E2 1486.551} C_VEL
LIN {X 0,Y 739.189,Z 845.935,A -85,B 0,C 180,E1 1492.437,E2 1492.437} C_VEL
LIN {X 0,Y 743.238,Z 857.523,A -85,B 0,C 180,E1 1492.814,E2 1492.814} C_VEL
LIN {X 0,Y 743.47,Z 946.188,A -85,B 0,C 180,E1 1494.322,E2 1494.322} C_VEL
LIN {X 0,Y 742.714,Z 1021.122,A -85,B 0,C 180,E1 1496.88,E2 1496.88} C_VEL
LIN {X 0,Y 741.482,Z 1091.628,A -85,B 0,C 180,E1 1500.606,E2 1500.606} C_VEL
LIN {X 0,Y 740.243,Z 1154.59,A -85,B 0,C 180,E1 1505.368,E2 1505.368} C_VEL
LIN {X 0,Y 739.47,Z 1202.967,A -85,B 0,C 180,E1 1510.455,E2 1510.455} C_VEL
LIN {X 0,Y 739.097,Z 1238.69,A -85,B 0,C 180,E1 1515.746,E2 1515.746} C_VEL
LIN {X 0,Y 739.093,Z 1262.394,A -85,B 0,C 180,E1 1521.148,E2 1521.148} C_VEL
LIN {X 0,Y 739.493,Z 1273.904,A -85,B 0,C 180,E1 1525.884,E2 1525.884} C_VEL
LIN {X 0,Y 739.256,Z 1276.339,A -85,B 0,C 180,E1 1531.763,E2 1531.763} C_VEL
LIN {X 0,Y 739.381,Z 1265.897,A -85,B 0,C 180,E1 1537.662,E2 1537.662} C_VEL
LIN {X 0,Y 739.399,Z 1241.418,A -85,B 0,C 180,E1 1543.643,E2 1543.643} C_VEL
LIN {X 0,Y 739.766,Z 1203.27,A -85,B 0,C 180,E1 1549.408,E2 1549.408} C_VEL
LIN {X 0,Y 740.539,Z 1151.4,A -85,B 0,C 180,E1 1554.823,E2 1554.823} C_VEL
LIN {X 0,Y 741.619,Z 1088.584,A -85,B 0,C 180,E1 1559.492,E2 1559.492} C_VEL
LIN {X 0,Y 742.815,Z 1018.796,A -85,B 0,C 180,E1 1563.125,E2 1563.125} C_VEL
LIN {X 0,Y 743.632,Z 944.044,A -85,B 0,C 180,E1 1565.636,E2 1565.636} C_VEL
LIN {X 0,Y 741.909,Z 850.185,A -85,B 0,C 180,E1 1567.261,E2 1567.261} C_VEL
LIN {X 0,Y 738.996,Z 844.06,A -85,B 0,C 180,E1 1567.544,E2 1567.544} C_VEL
LIN {X 0,Y 738.711,Z 844.06,A -85,B 0,C 180,E1 1576.505,E2 1576.505} C_VEL
LIN {X 0,Y 738.731,Z 844.06,A -85,B 0,C 180,E1 1584.183,E2 1584.183} C_VEL
LIN {X 0,Y 739.03,Z 844.06,A -85,B 0,C 180,E1 1591.137,E2 1591.137} C_VEL
LIN {X 0,Y 738.969,Z 844.06,A -85,B 0,C 180,E1 1599.03,E2 1599.03} C_VEL
LIN {X 0,Y 739.378,Z 844.06,A -85,B 0,C 180,E1 1607.539,E2 1607.539} C_VEL
LIN {X 0,Y 739.728,Z 844.06,A -85,B 0,C 180,E1 1617.042,E2 1617.042} C_VEL
LIN {X 0,Y 739.281,Z 844.06,A -85,B 0,C 180,E1 1624.672,E2 1624.672} C_VEL
LIN {X 0,Y 730.306,Z 844.06,A -85,B 0,C 180,E1 1627.351,E2 1627.351} C_VEL
LIN {X 0,Y 730.735,Z 844.06,A -85,B 0,C 180,E1 1633.793,E2 1633.793} C_VEL
LIN {X 0,Y 730.847,Z 844.06,A -85,B 0,C 180,E1 1641.279,E2 1641.279} C_VEL
LIN {X 0,Y 731.033,Z 844.06,A -85,B 0,C 180,E1 1649.165,E2 1649.165} C_VEL
LIN {X 0,Y 730.691,Z 844.06,A -85,B 0,C 180,E1 1657.744,E2 1657.744} C_VEL
LIN {X 0,Y 730.854,Z 844.06,A -85,B 0,C 180,E1 1665.962,E2 1665.962} C_VEL
LIN {X 0,Y 730.809,Z 845.831,A -85,B 0,C 180,E1 1671.853,E2 1671.853} C_VEL
LIN {X 0,Y 737.293,Z 860.391,A -85,B 0,C 180,E1 1672.423,E2 1672.423} C_VEL
LIN {X 0,Y 736.951,Z 953.671,A -85,B 0,C 180,E1 1673.936,E2 1673.936} C_VEL
LIN {X 0,Y 735.694,Z 1031.089,A -85,B 0,C 180,E1 1676.566,E2 1676.566} C_VEL
LIN {X 0,Y 734.31,Z 1102.256,A -85,B 0,C 180,E1 1680.378,E2 1680.378} C_VEL
LIN {X 0,Y 733.083,Z 1163.61,A -85,B 0,C 180,E1 1685.066,E2 1685.066} C_VEL
LIN {X 0,Y 732.143,Z 1214.964,A -85,B 0,C 180,E1 1690.554,E2 1690.554} C_VEL
LIN {X 0,Y 731.476,Z 1253.394,A -85,B 0,C 180,E1 1696.549,E2 1696.549} C_VEL
LIN {X 0,Y 731.38,Z 1276.024,A -85,B 0,C 180,E1 1702.254,E2 1702.254} C_VEL
LIN {X 0,Y 731.134,Z 1286.379,A -85,B 0,C 180,E1 1708.217,E2 1708.217} C_VEL
LIN {X 0,Y 731.301,Z 1283.831,A -85,B 0,C 180,E1 1714.162,E2 1714.162} C_VEL
LIN {X 0,Y 731.247,Z 1267.992,A -85,B 0,C 180,E1 1720.153,E2 1720.153} C_VEL
LIN {X 0,Y 731.477,Z 1238.889,A -85,B 0,C 180,E1 1726.038,E2 1726.038} C_VEL
LIN {X 0,Y 732.042,Z 1195.493,A -85,B 0,C 180,E1 1731.775,E2 1731.775} C_VEL
LIN {X 0,Y 733.21,Z 1138.958,A -85,B 0,C 180,E1 1737.018,E2 1737.018} C_VEL
LIN {X 0,Y 734.895,Z 1071.9,A -85,B 0,C 180,E1 1741.426,E2 1741.426} C_VEL
LIN {X 0,Y 736.466,Z 1000.336,A -85,B 0,C 180,E1 1744.631,E2 1744.631} C_VEL
LIN {X 0,Y 737.525,Z 927.653,A -85,B 0,C 180,E1 1746.619,E2 1746.619} C_VEL
LIN {X 0,Y 735.634,Z 854.031,A -85,B 0,C 180,E1 1747.754,E2 1747.754} C_VEL
LIN {X 0,Y 730.979,Z 844.06,A -85,B 0,C 180,E1 1748.314,E2 1748.314} C_VEL
LIN {X 0,Y 730.416,Z 844.06,A -85,B 0,C 180,E1 1754.258,E2 1754.258} C_VEL
LIN {X 0,Y 730.777,Z 844.06,A -85,B 0,C 180,E1 1762.262,E2 1762.262} C_VEL
LIN {X 0,Y 730.864,Z 844.06,A -85,B 0,C 180,E1 1768.065,E2 1768.065} C_VEL
LIN {X 0,Y 730.779,Z 844.06,A -85,B 0,C 180,E1 1774.835,E2 1774.835} C_VEL
LIN {X 0,Y 731.124,Z 844.06,A -85,B 0,C 180,E1 1782.511,E2 1782.511} C_VEL
LIN {X 0,Y 730.742,Z 844.06,A -85,B 0,C 180,E1 1791.062,E2 1791.062} C_VEL
LIN {X 0,Y 731.076,Z 844.06,A -85,B 0,C 180,E1 1798.236,E2 1798.236} C_VEL
LIN {X 0,Y 731.261,Z 844.06,A -85,B 0,C 180,E1 1805.376,E2 1805.376} C_VEL
LIN {X 0,Y 730.663,Z 844.06,A -85,B 0,C 180,E1 1813.834,E2 1813.834} C_VEL
LIN {X 0,Y 730.812,Z 844.06,A -85,B 0,C 180,E1 1821.322,E2 1821.322} C_VEL
LIN {X 0,Y 731,Z 844.06,A -85,B 0,C 180,E1 1829.211,E2 1829.211} C_VEL
LIN {X 0,Y 730.682,Z 844.06,A -85,B 0,C 180,E1 1837.793,E2 1837.793} C_VEL
LIN {X 0,Y 730.916,Z 844.06,A -85,B 0,C 180,E1 1845.967,E2 1845.967} C_VEL
LIN {X 0,Y 730.889,Z 845.877,A -85,B 0,C 180,E1 1851.935,E2 1851.935} C_VEL
LIN {X 0,Y 736.943,Z 860.77,A -85,B 0,C 180,E1 1852.482,E2 1852.482} C_VEL
LIN {X 0,Y 736.884,Z 947.425,A -85,B 0,C 180,E1 1853.987,E2 1853.987} C_VEL
LIN {X 0,Y 735.756,Z 1023.19,A -85,B 0,C 180,E1 1856.622,E2 1856.622} C_VEL
LIN {X 0,Y 734.101,Z 1094.134,A -85,B 0,C 180,E1 1860.45,E2 1860.45} C_VEL
LIN {X 0,Y 732.598,Z 1156.128,A -85,B 0,C 180,E1 1865.236,E2 1865.236} C_VEL
LIN {X 0,Y 731.616,Z 1204.333,A -85,B 0,C 180,E1 1870.413,E2 1870.413} C_VEL
LIN {X 0,Y 731.076,Z 1240.323,A -85,B 0,C 180,E1 1875.893,E2 1875.893} C_VEL
LIN {X 0,Y 731.143,Z 1262.393,A -85,B 0,C 180,E1 1881.051,E2 1881.051} C_VEL
LIN {X 0,Y 731.52,Z 1273.903,A -85,B 0,C 180,E1 1885.839,E2 1885.839} C_VEL
LIN {X 0,Y 731.262,Z 1276.34,A -85,B 0,C 180,E1 1891.783,E2 1891.783} C_VEL
LIN {X 0,Y 731.336,Z 1265.899,A -85,B 0,C 180,E1 1897.746,E2 1897.746} C_VEL
LIN {X 0,Y 731.383,Z 1241.422,A -85,B 0,C 180,E1 1903.795,E2 1903.795} C_VEL
LIN {X 0,Y 731.859,Z 1203.208,A -85,B 0,C 180,E1 1909.635,E2 1909.635} C_VEL
LIN {X 0,Y 732.891,Z 1151.407,A -85,B 0,C 180,E1 1915.1,E2 1915.1} C_VEL
LIN {X 0,Y 734.332,Z 1088.595,A -85,B 0,C 180,E1 1919.814,E2 1919.814} C_VEL
LIN {X 0,Y 735.934,Z 1018.768,A -85,B 0,C 180,E1 1923.478,E2 1923.478} C_VEL
LIN {X 0,Y 737.092,Z 944.066,A -85,B 0,C 180,E1 1926.001,E2 1926.001} C_VEL
LIN {X 0,Y 735.11,Z 853.422,A -85,B 0,C 180,E1 1927.627,E2 1927.627} C_VEL
LIN {X 0,Y 730.682,Z 844.06,A -85,B 0,C 180,E1 1928.044,E2 1928.044} C_VEL
LIN {X 0,Y 730.912,Z 844.06,A -85,B 0,C 180,E1 1935.922,E2 1935.922} C_VEL
LIN {X 0,Y 730.804,Z 844.06,A -85,B 0,C 180,E1 1943.704,E2 1943.704} C_VEL
LIN {X 0,Y 730.643,Z 844.06,A -85,B 0,C 180,E1 1952.128,E2 1952.128} C_VEL
LIN {X 0,Y 731.03,Z 844.06,A -85,B 0,C 180,E1 1958.685,E2 1958.685} C_VEL
LIN {X 0,Y 731.398,Z 844.06,A -85,B 0,C 180,E1 1967.401,E2 1967.401} C_VEL
LIN {X 0,Y 731.717,Z 844.06,A -85,B 0,C 180,E1 1977.01,E2 1977.01} C_VEL
LIN {X 0,Y 731.279,Z 844.06,A -85,B 0,C 180,E1 1985.337,E2 1985.337} C_VEL
LIN {X 0,Y 730.306,Z 844.06,A -85,B 0,C 180,E1 1987.351,E2 1987.351} C_VEL
LIN {X 0,Y 722.479,Z 844.06,A -85,B 0,C 180,E1 1990.084,E2 1990.084} C_VEL
LIN {X 0,Y 722.238,Z 844.06,A -85,B 0,C 180,E1 1995.202,E2 1995.202} C_VEL
LIN {X 0,Y 722.685,Z 844.06,A -85,B 0,C 180,E1 2001.531,E2 2001.531} C_VEL
LIN {X 0,Y 722.838,Z 844.06,A -85,B 0,C 180,E1 2009.529,E2 2009.529} C_VEL
LIN {X 0,Y 722.411,Z 844.06,A -85,B 0,C 180,E1 2018.254,E2 2018.254} C_VEL
LIN {X 0,Y 722.639,Z 844.06,A -85,B 0,C 180,E1 2026.379,E2 2026.379} C_VEL
LIN {X 0,Y 722.545,Z 845.878,A -85,B 0,C 180,E1 2031.337,E2 2031.337} C_VEL
LIN {X 0,Y 730.991,Z 863.424,A -85,B 0,C 180,E1 2032.079,E2 2032.079} C_VEL
LIN {X 0,Y 730.408,Z 954.777,A -85,B 0,C 180,E1 2033.591,E2 2033.591} C_VEL
LIN {X 0,Y 728.812,Z 1031.809,A -85,B 0,C 180,E1 2036.242,E2 2036.242} C_VEL
LIN {X 0,Y 727.068,Z 1101.568,A -85,B 0,C 180,E1 2040.006,E2 2040.006} C_VEL
LIN {X 0,Y 725.462,Z 1163.18,A -85,B 0,C 180,E1 2044.746,E2 2044.746} C_VEL
LIN {X 0,Y 724.372,Z 1214.966,A -85,B 0,C 180,E1 2050.337,E2 2050.337} C_VEL
LIN {X 0,Y 723.594,Z 1253.21,A -85,B 0,C 180,E1 2056.363,E2 2056.363} C_VEL
LIN {X 0,Y 723.416,Z 1276.024,A -85,B 0,C 180,E1 2062.168,E2 2062.168} C_VEL
LIN {X 0,Y 723.138,Z 1286.379,A -85,B 0,C 180,E1 2068.197,E2 2068.197} C_VEL
LIN {X 0,Y 723.271,Z 1283.831,A -85,B 0,C 180,E1 2074.208,E2 2074.208} C_VEL
LIN {X 0,Y 723.197,Z 1267.993,A -85,B 0,C 180,E1 2080.267,E2 2080.267} C_VEL
LIN {X 0,Y 723.486,Z 1238.753,A -85,B 0,C 180,E1 2086.242,E2 2086.242} C_VEL
LIN {X 0,Y 724.266,Z 1195.871,A -85,B 0,C 180,E1 2091.98,E2 2091.98} C_VEL
LIN {X 0,Y 725.695,Z 1140.087,A -85,B 0,C 180,E1 2097.23,E2 2097.23} C_VEL
LIN {X 0,Y 727.756,Z 1073.617,A -85,B 0,C 180,E1 2101.671,E2 2101.671} C_VEL
LIN {X 0,Y 729.68,Z 1002.576,A -85,B 0,C 180,E1 2104.915,E2 2104.915} C_VEL
LIN {X 0,Y 731.065,Z 928.881,A -85,B 0,C 180,E1 2106.972,E2 2106.972} C_VEL
LIN {X 0,Y 729.594,Z 857.788,A -85,B 0,C 180,E1 2108.076,E2 2108.076} C_VEL
LIN {X 0,Y 722.897,Z 844.06,A -85,B 0,C 180,E1 2108.823,E2 2108.823} C_VEL
LIN {X 0,Y 722.08,Z 844.06,A -85,B 0,C 180,E1 2115.294,E2 2115.294} C_VEL
LIN {X 0,Y 722.879,Z 844.06,A -85,B 0,C 180,E1 2121.88,E2 2121.88} C_VEL
LIN {X 0,Y 722.526,Z 844.06,A -85,B 0,C 180,E1 2129.065,E2 2129.065} C_VEL
LIN {X 0,Y 722.3,Z 844.06,A -85,B 0,C 180,E1 2135.969,E2 2135.969} C_VEL
LIN {X 0,Y 722.568,Z 844.06,A -85,B 0,C 180,E1 2143.555,E2 2143.555} C_VEL
LIN {X 0,Y 722.798,Z 844.06,A -85,B 0,C 180,E1 2150.963,E2 2150.963} C_VEL
LIN {X 0,Y 723.08,Z 844.06,A -85,B 0,C 180,E1 2158.216,E2 2158.216} C_VEL
LIN {X 0,Y 723.233,Z 844.06,A -85,B 0,C 180,E1 2165.436,E2 2165.436} C_VEL
LIN {X 0,Y 722.584,Z 844.06,A -85,B 0,C 180,E1 2173.991,E2 2173.991} C_VEL
LIN {X 0,Y 722.672,Z 844.06,A -85,B 0,C 180,E1 2181.574,E2 2181.574} C_VEL
LIN {X 0,Y 722.794,Z 844.06,A -85,B 0,C 180,E1 2189.575,E2 2189.575} C_VEL
LIN {X 0,Y 722.436,Z 844.06,A -85,B 0,C 180,E1 2198.302,E2 2198.302} C_VEL
LIN {X 0,Y 722.689,Z 844.06,A -85,B 0,C 180,E1 2206.431,E2 2206.431} C_VEL
LIN {X 0,Y 722.62,Z 845.929,A -85,B 0,C 180,E1 2211.422,E2 2211.422} C_VEL
LIN {X 0,Y 730.614,Z 862.926,A -85,B 0,C 180,E1 2212.127,E2 2212.127} C_VEL
LIN {X 0,Y 730.301,Z 949.286,A -85,B 0,C 180,E1 2213.662,E2 2213.662} C_VEL
LIN {X 0,Y 728.793,Z 1025.266,A -85,B 0,C 180,E1 2216.359,E2 2216.359} C_VEL
LIN {X 0,Y 726.807,Z 1095.381,A -85,B 0,C 180,E1 2220.209,E2 2220.209} C_VEL
LIN {X 0,Y 725.006,Z 1156.968,A -85,B 0,C 180,E1 2225.038,E2 2225.038} C_VEL
LIN {X 0,Y 723.76,Z 1205.334,A -85,B 0,C 180,E1 2230.323,E2 2230.323} C_VEL
LIN {X 0,Y 723.203,Z 1240.322,A -85,B 0,C 180,E1 2235.736,E2 2235.736} C_VEL
LIN {X 0,Y 723.22,Z 1262.392,A -85,B 0,C 180,E1 2240.952,E2 2240.952} C_VEL
LIN {X 0,Y 723.528,Z 1273.902,A -85,B 0,C 180,E1 2245.793,E2 2245.793} C_VEL
LIN {X 0,Y 723.255,Z 1276.341,A -85,B 0,C 180,E1 2251.802,E2 2251.802} C_VEL
LIN {X 0,Y 723.292,Z 1265.9,A -85,B 0,C 180,E1 2257.833,E2 2257.833} C_VEL
LIN {X 0,Y 723.375,Z 1241.426,A -85,B 0,C 180,E1 2263.951,E2 2263.951} C_VEL
LIN {X 0,Y 723.997,Z 1204.026,A -85,B 0,C 180,E1 2269.751,E2 2269.751} C_VEL
LIN {X 0,Y 725.251,Z 1152.808,A -85,B 0,C 180,E1 2275.252,E2 2275.252} C_VEL
LIN {X 0,Y 727.042,Z 1090.39,A -85,B 0,C 180,E1 2280.03,E2 2280.03} C_VEL
LIN {X 0,Y 729.064,Z 1019.471,A -85,B 0,C 180,E1 2283.806,E2 2283.806} C_VEL
LIN {X 0,Y 730.557,Z 943.929,A -85,B 0,C 180,E1 2286.378,E2 2286.378} C_VEL
LIN {X 0,Y 728.693,Z 856.212,A -85,B 0,C 180,E1 2287.983,E2 2287.983} C_VEL
LIN {X 0,Y 722.418,Z 844.06,A -85,B 0,C 180,E1 2288.558,E2 2288.558} C_VEL
LIN {X 0,Y 722.717,Z 844.06,A -85,B 0,C 180,E1 2296.381,E2 2296.381} C_VEL
LIN {X 0,Y 722.717,Z 844.06,A -85,B 0,C 180,E1 2303.889,E2 2303.889} C_VEL
LIN {X 0,Y 722.769,Z 844.06,A -85,B 0,C 180,E1 2311.797,E2 2311.797} C_VEL
LIN {X 0,Y 722.613,Z 844.06,A -85,B 0,C 180,E1 2319.712,E2 2319.712} C_VEL
LIN {X 0,Y 723.384,Z 844.06,A -85,B 0,C 180,E1 2327.259,E2 2327.259} C_VEL
LIN {X 0,Y 723.676,Z 844.06,A -85,B 0,C 180,E1 2336.976,E2 2336.976} C_VEL
LIN {X 0,Y 723.227,Z 844.06,A -85,B 0,C 180,E1 2345.397,E2 2345.397} C_VEL
LIN {X 0,Y 722.479,Z 844.06,A -85,B 0,C 180,E1 2350.084,E2 2350.084} C_VEL
LIN {X 0,Y 715.227,Z 844.06,A -85,B 0,C 180,E1 2352.86,E2 2352.86} C_VEL
LIN {X 0,Y 714.535,Z 844.06,A -85,B 0,C 180,E1 2361.79,E2 2361.79} C_VEL
LIN {X 0,Y 714.639,Z 844.06,A -85,B 0,C 180,E1 2369.902,E2 2369.902} C_VEL
LIN {X 0,Y 714.676,Z 844.06,A -85,B 0,C 180,E1 2377.274,E2 2377.274} C_VEL
LIN {X 0,Y 714.627,Z 844.06,A -85,B 0,C 180,E1 2386.394,E2 2386.394} C_VEL
LIN {X 0,Y 714.25,Z 845.347,A -85,B 0,C 180,E1 2390.796,E2 2390.796} C_VEL
LIN {X 0,Y 724.703,Z 866.593,A -85,B 0,C 180,E1 2391.73,E2 2391.73} C_VEL
LIN {X 0,Y 723.873,Z 955.961,A -85,B 0,C 180,E1 2393.241,E2 2393.241} C_VEL
LIN {X 0,Y 721.966,Z 1032.509,A -85,B 0,C 180,E1 2395.912,E2 2395.912} C_VEL
LIN {X 0,Y 719.842,Z 1101.835,A -85,B 0,C 180,E1 2399.692,E2 2399.692} C_VEL
LIN {X 0,Y 717.893,Z 1163.011,A -85,B 0,C 180,E1 2404.444,E2 2404.444} C_VEL
LIN {X 0,Y 716.636,Z 1214.298,A -85,B 0,C 180,E1 2410.027,E2 2410.027} C_VEL
LIN {X 0,Y 715.712,Z 1253.21,A -85,B 0,C 180,E1 2416.209,E2 2416.209} C_VEL
LIN {X 0,Y 715.447,Z 1276.024,A -85,B 0,C 180,E1 2422.08,E2 2422.08} C_VEL
LIN {X 0,Y 715.158,Z 1286.379,A -85,B 0,C 180,E1 2428.177,E2 2428.177} C_VEL
LIN {X 0,Y 715.257,Z 1283.831,A -85,B 0,C 180,E1 2434.256,E2 2434.256} C_VEL
LIN {X 0,Y 715.18,Z 1267.994,A -85,B 0,C 180,E1 2440.384,E2 2440.384} C_VEL
LIN {X 0,Y 715.561,Z 1239.677,A -85,B 0,C 180,E1 2446.277,E2 2446.277} C_VEL
LIN {X 0,Y 716.497,Z 1197.427,A -85,B 0,C 180,E1 2452.056,E2 2452.056} C_VEL
LIN {X 0,Y 718.205,Z 1141.748,A -85,B 0,C 180,E1 2457.403,E2 2457.403} C_VEL
LIN {X 0,Y 720.646,Z 1074.711,A -85,B 0,C 180,E1 2461.957,E2 2461.957} C_VEL
LIN {X 0,Y 722.968,Z 1002.832,A -85,B 0,C 180,E1 2465.278,E2 2465.278} C_VEL
LIN {X 0,Y 724.618,Z 930.882,A -85,B 0,C 180,E1 2467.316,E2 2467.316} C_VEL
LIN {X 0,Y 723.13,Z 860.353,A -85,B 0,C 180,E1 2468.446,E2 2468.446} C_VEL
LIN {X 0,Y 714.883,Z 844.06,A -85,B 0,C 180,E1 2469.267,E2 2469.267} C_VEL
LIN {X 0,Y 714.009,Z 844.06,A -85,B 0,C 180,E1 2476.356,E2 2476.356} C_VEL
LIN {X 0,Y 714.663,Z 844.06,A -85,B 0,C 180,E1 2482.798,E2 2482.798} C_VEL
LIN {X 0,Y 714.395,Z 844.06,A -85,B 0,C 180,E1 2490.087,E2 2490.087} C_VEL
LIN {X 0,Y 714.026,Z 844.06,A -85,B 0,C 180,E1 2496.877,E2 2496.877} C_VEL
LIN {X 0,Y 714.658,Z 844.06,A -85,B 0,C 180,E1 2503.368,E2 2503.368} C_VEL
LIN {X 0,Y 714.822,Z 844.06,A -85,B 0,C 180,E1 2510.861,E2 2510.861} C_VEL
LIN {X 0,Y 715.083,Z 844.06,A -85,B 0,C 180,E1 2518.196,E2 2518.196} C_VEL
LIN {X 0,Y 715.18,Z 844.06,A -85,B 0,C 180,E1 2525.497,E2 2525.497} C_VEL
LIN {X 0,Y 715.188,Z 844.06,A -85,B 0,C 180,E1 2532.889,E2 2532.889} C_VEL
LIN {X 0,Y 714.521,Z 844.06,A -85,B 0,C 180,E1 2541.832,E2 2541.832} C_VEL
LIN {X 0,Y 714.586,Z 844.06,A -85,B 0,C 180,E1 2549.95,E2 2549.95} C_VEL
LIN {X 0,Y 714.708,Z 844.06,A -85,B 0,C 180,E1 2557.278,E2 2557.278} C_VEL
LIN {X 0,Y 714.702,Z 844.06,A -85,B 0,C 180,E1 2566.4,E2 2566.4} C_VEL
LIN {X 0,Y 714.356,Z 845.66,A -85,B 0,C 180,E1 2570.888,E2 2570.888} C_VEL
LIN {X 0,Y 724.373,Z 866.327,A -85,B 0,C 180,E1 2571.784,E2 2571.784} C_VEL
LIN {X 0,Y 723.734,Z 951.104,A -85,B 0,C 180,E1 2573.331,E2 2573.331} C_VEL
LIN {X 0,Y 721.858,Z 1027.439,A -85,B 0,C 180,E1 2576.097,E2 2576.097} C_VEL
LIN {X 0,Y 719.416,Z 1098.499,A -85,B 0,C 180,E1 2580.089,E2 2580.089} C_VEL
LIN {X 0,Y 717.312,Z 1159.438,A -85,B 0,C 180,E1 2584.986,E2 2584.986} C_VEL
LIN {X 0,Y 715.909,Z 1206.948,A -85,B 0,C 180,E1 2590.311,E2 2590.311} C_VEL
LIN {X 0,Y 715.306,Z 1240.436,A -85,B 0,C 180,E1 2595.598,E2 2595.598} C_VEL
LIN {X 0,Y 715.035,Z 1264.334,A -85,B 0,C 180,E1 2601.462,E2 2601.462} C_VEL
LIN {X 0,Y 714.96,Z 1275.393,A -85,B 0,C 180,E1 2606.96,E2 2606.96} C_VEL
LIN {X 0,Y 715.038,Z 1275.317,A -85,B 0,C 180,E1 2613.039,E2 2613.039} C_VEL
LIN {X 0,Y 715.027,Z 1264.049,A -85,B 0,C 180,E1 2618.538,E2 2618.538} C_VEL
LIN {X 0,Y 715.299,Z 1240.226,A -85,B 0,C 180,E1 2624.354,E2 2624.354} C_VEL
LIN {X 0,Y 716.093,Z 1202.511,A -85,B 0,C 180,E1 2630.179,E2 2630.179} C_VEL
LIN {X 0,Y 717.623,Z 1151.421,A -85,B 0,C 180,E1 2635.672,E2 2635.672} C_VEL
LIN {X 0,Y 719.798,Z 1088.397,A -85,B 0,C 180,E1 2640.493,E2 2640.493} C_VEL
LIN {X 0,Y 722.258,Z 1018.131,A -85,B 0,C 180,E1 2644.227,E2 2644.227} C_VEL
LIN {X 0,Y 724.133,Z 942.957,A -85,B 0,C 180,E1 2646.781,E2 2646.781} C_VEL
LIN {X 0,Y 722.132,Z 859.299,A -85,B 0,C 180,E1 2648.353,E2 2648.353} C_VEL
LIN {X 0,Y 714.196,Z 844.06,A -85,B 0,C 180,E1 2649.137,E2 2649.137} C_VEL
LIN {X 0,Y 714.727,Z 844.06,A -85,B 0,C 180,E1 2656.357,E2 2656.357} C_VEL
LIN {X 0,Y 714.454,Z 844.06,A -85,B 0,C 180,E1 2664.808,E2 2664.808} C_VEL
LIN {X 0,Y 714.777,Z 844.06,A -85,B 0,C 180,E1 2671.703,E2 2671.703} C_VEL
LIN {X 0,Y 714.703,Z 844.06,A -85,B 0,C 180,E1 2679.478,E2 2679.478} C_VEL
LIN {X 0,Y 715.407,Z 844.06,A -85,B 0,C 180,E1 2687.115,E2 2687.115} C_VEL
LIN {X 0,Y 715.635,Z 844.06,A -85,B 0,C 180,E1 2696.942,E2 2696.942} C_VEL
LIN {X 0,Y 715.178,Z 844.06,A -85,B 0,C 180,E1 2705.458,E2 2705.458} C_VEL
LIN {X 0,Y 715.227,Z 844.06,A -85,B 0,C 180,E1 2712.86,E2 2712.86} C_VEL
LIN {X 0,Y 706.161,Z 844.06,A -85,B 0,C 180,E1 2715.623,E2 2715.623} C_VEL
LIN {X 0,Y 706.422,Z 844.06,A -85,B 0,C 180,E1 2722.053,E2 2722.053} C_VEL
LIN {X 0,Y 706.471,Z 844.06,A -85,B 0,C 180,E1 2730.283,E2 2730.283} C_VEL
LIN {X 0,Y 706.254,Z 844.06,A -85,B 0,C 180,E1 2738.394,E2 2738.394} C_VEL
LIN {X 0,Y 706.693,Z 844.06,A -85,B 0,C 180,E1 2745.954,E2 2745.954} C_VEL
LIN {X 0,Y 706.212,Z 845.848,A -85,B 0,C 180,E1 2750.268,E2 2750.268} C_VEL
LIN {X 0,Y 718.428,Z 870.645,A -85,B 0,C 180,E1 2751.385,E2 2751.385} C_VEL
LIN {X 0,Y 717.313,Z 957.774,A -85,B 0,C 180,E1 2752.899,E2 2752.899} C_VEL
LIN {X 0,Y 715.085,Z 1033.997,A -85,B 0,C 180,E1 2755.61,E2 2755.61} C_VEL
LIN {X 0,Y 712.585,Z 1102.913,A -85,B 0,C 180,E1 2759.426,E2 2759.426} C_VEL
LIN {X 0,Y 710.299,Z 1163.609,A -85,B 0,C 180,E1 2764.208,E2 2764.208} C_VEL
LIN {X 0,Y 708.801,Z 1215.428,A -85,B 0,C 180,E1 2769.948,E2 2769.948} C_VEL
LIN {X 0,Y 707.834,Z 1253.211,A -85,B 0,C 180,E1 2776.053,E2 2776.053} C_VEL
LIN {X 0,Y 707.202,Z 1277.662,A -85,B 0,C 180,E1 2782.607,E2 2782.607} C_VEL
LIN {X 0,Y 707.162,Z 1286.379,A -85,B 0,C 180,E1 2788.157,E2 2788.157} C_VEL
LIN {X 0,Y 707.225,Z 1283.735,A -85,B 0,C 180,E1 2794.366,E2 2794.366} C_VEL
LIN {X 0,Y 707.132,Z 1267.995,A -85,B 0,C 180,E1 2800.503,E2 2800.503} C_VEL
LIN {X 0,Y 707.596,Z 1239.48,A -85,B 0,C 180,E1 2806.498,E2 2806.498} C_VEL
LIN {X 0,Y 708.75,Z 1197.68,A -85,B 0,C 180,E1 2812.281,E2 2812.281} C_VEL
LIN {X 0,Y 710.721,Z 1142.059,A -85,B 0,C 180,E1 2817.691,E2 2817.691} C_VEL
LIN {X 0,Y 713.584,Z 1075.298,A -85,B 0,C 180,E1 2822.277,E2 2822.277} C_VEL
LIN {X 0,Y 716.245,Z 1004.097,A -85,B 0,C 180,E1 2825.61,E2 2825.61} C_VEL
LIN {X 0,Y 718.238,Z 930.391,A -85,B 0,C 180,E1 2827.715,E2 2827.715} C_VEL
LIN {X 0,Y 716.826,Z 863.743,A -85,B 0,C 180,E1 2828.805,E2 2828.805} C_VEL
LIN {X 0,Y 706.884,Z 844.06,A -85,B 0,C 180,E1 2829.88,E2 2829.88} C_VEL
LIN {X 0,Y 706.271,Z 844.06,A -85,B 0,C 180,E1 2837.799,E2 2837.799} C_VEL
LIN {X 0,Y 706.909,Z 844.06,A -85,B 0,C 180,E1 2845.365,E2 2845.365} C_VEL
LIN {X 0,Y 706.882,Z 844.06,A -85,B 0,C 180,E1 2853.922,E2 2853.922} C_VEL
LIN {X 0,Y 706.7,Z 844.06,A -85,B 0,C 180,E1 2863.175,E2 2863.175} C_VEL
LIN {X 0,Y 706.864,Z 844.06,A -85,B 0,C 180,E1 2870.758,E2 2870.758} C_VEL
LIN {X 0,Y 707.087,Z 844.06,A -85,B 0,C 180,E1 2878.176,E2 2878.176} C_VEL
LIN {X 0,Y 707.143,Z 844.06,A -85,B 0,C 180,E1 2885.56,E2 2885.56} C_VEL
LIN {X 0,Y 707.079,Z 844.06,A -85,B 0,C 180,E1 2893.04,E2 2893.04} C_VEL
LIN {X 0,Y 706.796,Z 844.06,A -85,B 0,C 180,E1 2901.036,E2 2901.036} C_VEL
LIN {X 0,Y 706.647,Z 844.06,A -85,B 0,C 180,E1 2909.638,E2 2909.638} C_VEL
LIN {X 0,Y 706.51,Z 844.06,A -85,B 0,C 180,E1 2917.756,E2 2917.756} C_VEL
LIN {X 0,Y 706.772,Z 844.06,A -85,B 0,C 180,E1 2926.005,E2 2926.005} C_VEL
LIN {X 0,Y 706.273,Z 845.836,A -85,B 0,C 180,E1 2930.356,E2 2930.356} C_VEL
LIN {X 0,Y 718.138,Z 870.154,A -85,B 0,C 180,E1 2931.44,E2 2931.44} C_VEL
LIN {X 0,Y 717.19,Z 952.607,A -85,B 0,C 180,E1 2932.985,E2 2932.985} C_VEL
LIN {X 0,Y 714.944,Z 1028.947,A -85,B 0,C 180,E1 2935.798,E2 2935.798} C_VEL
LIN {X 0,Y 712.154,Z 1099.38,A -85,B 0,C 180,E1 2939.814,E2 2939.814} C_VEL
LIN {X 0,Y 709.76,Z 1159.432,A -85,B 0,C 180,E1 2944.701,E2 2944.701} C_VEL
LIN {X 0,Y 708.061,Z 1207.736,A -85,B 0,C 180,E1 2950.189,E2 2950.189} C_VEL
LIN {X 0,Y 707.264,Z 1241.876,A -85,B 0,C 180,E1 2955.724,E2 2955.724} C_VEL
LIN {X 0,Y 707.088,Z 1264.333,A -85,B 0,C 180,E1 2961.365,E2 2961.365} C_VEL
LIN {X 0,Y 706.97,Z 1275.393,A -85,B 0,C 180,E1 2966.926,E2 2966.926} C_VEL
LIN {X 0,Y 707.028,Z 1275.317,A -85,B 0,C 180,E1 2973.074,E2 2973.074} C_VEL
LIN {X 0,Y 707.028,Z 1264.191,A -85,B 0,C 180,E1 2978.591,E2 2978.591} C_VEL
LIN {X 0,Y 707.33,Z 1240.347,A -85,B 0,C 180,E1 2984.496,E2 2984.496} C_VEL
LIN {X 0,Y 708.254,Z 1204.117,A -85,B 0,C 180,E1 2990.199,E2 2990.199} C_VEL
LIN {X 0,Y 709.998,Z 1153.196,A -85,B 0,C 180,E1 2995.798,E2 2995.798} C_VEL
LIN {X 0,Y 712.564,Z 1090.06,A -85,B 0,C 180,E1 3000.729,E2 3000.729} C_VEL
LIN {X 0,Y 715.429,Z 1019.455,A -85,B 0,C 180,E1 3004.543,E2 3004.543} C_VEL
LIN {X 0,Y 717.584,Z 945.116,A -85,B 0,C 180,E1 3007.113,E2 3007.113} C_VEL
LIN {X 0,Y 716.109,Z 863.003,A -85,B 0,C 180,E1 3008.689,E2 3008.689} C_VEL
LIN {X 0,Y 706.064,Z 844.06,A -85,B 0,C 180,E1 3009.624,E2 3009.624} C_VEL
LIN {X 0,Y 706.823,Z 844.06,A -85,B 0,C 180,E1 3015.953,E2 3015.953} C_VEL
LIN {X 0,Y 706.641,Z 844.06,A -85,B 0,C 180,E1 3023.792,E2 3023.792} C_VEL
LIN {X 0,Y 706.815,Z 844.06,A -85,B 0,C 180,E1 3031.101,E2 3031.101} C_VEL
LIN {X 0,Y 706.737,Z 844.06,A -85,B 0,C 180,E1 3039.236,E2 3039.236} C_VEL
LIN {X 0,Y 707.398,Z 844.06,A -85,B 0,C 180,E1 3047.275,E2 3047.275} C_VEL
LIN {X 0,Y 707.591,Z 844.06,A -85,B 0,C 180,E1 3056.916,E2 3056.916} C_VEL
LIN {X 0,Y 707.136,Z 844.06,A -85,B 0,C 180,E1 3065.52,E2 3065.52} C_VEL
LIN {X 0,Y 707.148,Z 844.06,A -85,B 0,C 180,E1 3072.997,E2 3072.997} C_VEL
LIN {X 0,Y 706.161,Z 844.06,A -85,B 0,C 180,E1 3075.623,E2 3075.623} C_VEL
LIN {X 0,Y 698.55,Z 844.06,A -85,B 0,C 180,E1 3078.447,E2 3078.447} C_VEL
LIN {X 0,Y 698.365,Z 844.06,A -85,B 0,C 180,E1 3086.421,E2 3086.421} C_VEL
LIN {X 0,Y 698.112,Z 844.06,A -85,B 0,C 180,E1 3093.626,E2 3093.626} C_VEL
LIN {X 0,Y 697.839,Z 844.06,A -85,B 0,C 180,E1 3099.862,E2 3099.862} C_VEL
LIN {X 0,Y 698.362,Z 844.06,A -85,B 0,C 180,E1 3106.84,E2 3106.84} C_VEL
LIN {X 0,Y 698.134,Z 845.807,A -85,B 0,C 180,E1 3109.714,E2 3109.714} C_VEL
LIN {X 0,Y 712.187,Z 871.986,A -85,B 0,C 180,E1 3110.999,E2 3110.999} C_VEL
LIN {X 0,Y 710.89,Z 957.772,A -85,B 0,C 180,E1 3112.507,E2 3112.507} C_VEL
LIN {X 0,Y 708.289,Z 1034.154,A -85,B 0,C 180,E1 3115.241,E2 3115.241} C_VEL
LIN {X 0,Y 705.407,Z 1102.85,A -85,B 0,C 180,E1 3119.077,E2 3119.077} C_VEL
LIN {X 0,Y 702.729,Z 1163.663,A -85,B 0,C 180,E1 3123.915,E2 3123.915} C_VEL
LIN {X 0,Y 700.982,Z 1214.459,A -85,B 0,C 180,E1 3129.583,E2 3129.583} C_VEL
LIN {X 0,Y 699.935,Z 1253.213,A -85,B 0,C 180,E1 3135.892,E2 3135.892} C_VEL
LIN {X 0,Y 699.235,Z 1277.66,A -85,B 0,C 180,E1 3142.523,E2 3142.523} C_VEL
LIN {X 0,Y 699.182,Z 1286.379,A -85,B 0,C 180,E1 3148.135,E2 3148.135} C_VEL
LIN {X 0,Y 699.253,Z 1283.831,A -85,B 0,C 180,E1 3154.353,E2 3154.353} C_VEL
LIN {X 0,Y 699.132,Z 1267.996,A -85,B 0,C 180,E1 3160.625,E2 3160.625} C_VEL
LIN {X 0,Y 699.702,Z 1241.38,A -85,B 0,C 180,E1 3166.365,E2 3166.365} C_VEL
LIN {X 0,Y 700.941,Z 1200.117,A -85,B 0,C 180,E1 3172.248,E2 3172.248} C_VEL
LIN {X 0,Y 703.197,Z 1145.562,A -85,B 0,C 180,E1 3177.721,E2 3177.721} C_VEL
LIN {X 0,Y 706.375,Z 1079.692,A -85,B 0,C 180,E1 3182.384,E2 3182.384} C_VEL
LIN {X 0,Y 709.471,Z 1008.688,A -85,B 0,C 180,E1 3185.823,E2 3185.823} C_VEL
LIN {X 0,Y 711.76,Z 934.167,A -85,B 0,C 180,E1 3188.037,E2 3188.037} C_VEL
LIN {X 0,Y 710.673,Z 867.118,A -85,B 0,C 180,E1 3189.162,E2 3189.162} C_VEL
LIN {X 0,Y 698.935,Z 844.06,A -85,B 0,C 180,E1 3190.444,E2 3190.444} C_VEL
LIN {X 0,Y 698.912,Z 844.06,A -85,B 0,C 180,E1 3200.381,E2 3200.381} C_VEL
LIN {X 0,Y 698.775,Z 844.06,A -85,B 0,C 180,E1 3207.89,E2 3207.89} C_VEL
LIN {X 0,Y 698.571,Z 844.06,A -85,B 0,C 180,E1 3214.969,E2 3214.969} C_VEL
LIN {X 0,Y 698.78,Z 844.06,A -85,B 0,C 180,E1 3222.979,E2 3222.979} C_VEL
LIN {X 0,Y 698.816,Z 844.06,A -85,B 0,C 180,E1 3230.901,E2 3230.901} C_VEL
LIN {X 0,Y 699.11,Z 844.06,A -85,B 0,C 180,E1 3238.155,E2 3238.155} C_VEL
LIN {X 0,Y 699.091,Z 844.06,A -85,B 0,C 180,E1 3245.624,E2 3245.624} C_VEL
LIN {X 0,Y 698.979,Z 844.06,A -85,B 0,C 180,E1 3253.193,E2 3253.193} C_VEL
LIN {X 0,Y 698.81,Z 844.06,A -85,B 0,C 180,E1 3261.011,E2 3261.011} C_VEL
LIN {X 0,Y 698.747,Z 844.06,A -85,B 0,C 180,E1 3269.265,E2 3269.265} C_VEL
LIN {X 0,Y 698.309,Z 844.06,A -85,B 0,C 180,E1 3278.279,E2 3278.279} C_VEL
LIN {X 0,Y 698.443,Z 844.06,A -85,B 0,C 180,E1 3286.846,E2 3286.846} C_VEL
LIN {X 0,Y 698.166,Z 845.834,A -85,B 0,C 180,E1 3289.804,E2 3289.804} C_VEL
LIN {X 0,Y 711.943,Z 873.652,A -85,B 0,C 180,E1 3291.087,E2 3291.087} C_VEL
LIN {X 0,Y 710.67,Z 955.306,A -85,B 0,C 180,E1 3292.667,E2 3292.667} C_VEL
LIN {X 0,Y 708.102,Z 1029.999,A -85,B 0,C 180,E1 3295.473,E2 3295.473} C_VEL
LIN {X 0,Y 704.866,Z 1100.448,A -85,B 0,C 180,E1 3299.546,E2 3299.546} C_VEL
LIN {X 0,Y 702.104,Z 1161.181,A -85,B 0,C 180,E1 3304.577,E2 3304.577} C_VEL
LIN {X 0,Y 700.174,Z 1209.656,A -85,B 0,C 180,E1 3310.219,E2 3310.219} C_VEL
LIN {X 0,Y 699.252,Z 1243.432,A -85,B 0,C 180,E1 3315.878,E2 3315.878} C_VEL
LIN {X 0,Y 699.082,Z 1264.756,A -85,B 0,C 180,E1 3321.404,E2 3321.404} C_VEL
LIN {X 0,Y 698.999,Z 1275.392,A -85,B 0,C 180,E1 3326.891,E2 3326.891} C_VEL
LIN {X 0,Y 699.036,Z 1275.317,A -85,B 0,C 180,E1 3333.109,E2 3333.109} C_VEL
LIN {X 0,Y 698.956,Z 1263.471,A -85,B 0,C 180,E1 3338.925,E2 3338.925} C_VEL
LIN {X 0,Y 699.392,Z 1241.438,A -85,B 0,C 180,E1 3344.44,E2 3344.44} C_VEL
LIN {X 0,Y 700.407,Z 1205.345,A -85,B 0,C 180,E1 3350.27,E2 3350.27} C_VEL
LIN {X 0,Y 702.376,Z 1154.967,A -85,B 0,C 180,E1 3355.927,E2 3355.927} C_VEL
LIN {X 0,Y 705.238,Z 1092.809,A -85,B 0,C 180,E1 3360.889,E2 3360.889} C_VEL
LIN {X 0,Y 708.529,Z 1022.326,A -85,B 0,C 180,E1 3364.79,E2 3364.79} C_VEL
LIN {X 0,Y 711.034,Z 947.919,A -85,B 0,C 180,E1 3367.435,E2 3367.435} C_VEL
LIN {X 0,Y 710.176,Z 866.637,A -85,B 0,C 180,E1 3369.028,E2 3369.028} C_VEL
LIN {X 0,Y 697.97,Z 844.06,A -85,B 0,C 180,E1 3370.178,E2 3370.178} C_VEL
LIN {X 0,Y 698.509,Z 844.06,A -85,B 0,C 180,E1 3376.806,E2 3376.806} C_VEL
LIN {X 0,Y 698.374,Z 844.06,A -85,B 0,C 180,E1 3384.831,E2 3384.831} C_VEL
LIN {X 0,Y 698.542,Z 844.06,A -85,B 0,C 180,E1 3392.143,E2 3392.143} C_VEL
LIN {X 0,Y 698.796,Z 844.06,A -85,B 0,C 180,E1 3398.989,E2 3398.989} C_VEL
LIN {X 0,Y 699.449,Z 844.06,A -85,B 0,C 180,E1 3408.089,E2 3408.089} C_VEL
LIN {X 0,Y 699.153,Z 844.06,A -85,B 0,C 180,E1 3418.115,E2 3418.115} C_VEL
LIN {X 0,Y 699.088,Z 844.06,A -85,B 0,C 180,E1 3425.584,E2 3425.584} C_VEL
LIN {X 0,Y 699.045,Z 844.06,A -85,B 0,C 180,E1 3433.151,E2 3433.151} C_VEL
LIN {X 0,Y 698.55,Z 844.06,A -85,B 0,C 180,E1 3438.447,E2 3438.447} C_VEL
LIN {X 0,Y 690.67,Z 844.06,A -85,B 0,C 180,E1 3441.308,E2 3441.308} C_VEL
LIN {X 0,Y 690.552,Z 844.06,A -85,B 0,C 180,E1 3449.834,E2 3449.834} C_VEL
LIN {X 0,Y 690.535,Z 844.06,A -85,B 0,C 180,E1 3457.142,E2 3457.142} C_VEL
LIN {X 0,Y 690.437,Z 844.06,A -85,B 0,C 180,E1 3466.22,E2 3466.22} C_VEL
LIN {X 0,Y 689.989,Z 845.162,A -85,B 0,C 180,E1 3469.13,E2 3469.13} C_VEL
LIN {X 0,Y 705.976,Z 876.339,A -85,B 0,C 180,E1 3470.646,E2 3470.646} C_VEL
LIN {X 0,Y 704.311,Z 961.128,A -85,B 0,C 180,E1 3472.194,E2 3472.194} C_VEL
LIN {X 0,Y 701.335,Z 1038.03,A -85,B 0,C 180,E1 3475.039,E2 3475.039} C_VEL
LIN {X 0,Y 697.993,Z 1107.273,A -85,B 0,C 180,E1 3479.03,E2 3479.03} C_VEL
LIN {X 0,Y 694.983,Z 1168.962,A -85,B 0,C 180,E1 3484.124,E2 3484.124} C_VEL
LIN {X 0,Y 693.114,Z 1218.122,A -85,B 0,C 180,E1 3489.842,E2 3489.842} C_VEL
LIN {X 0,Y 691.883,Z 1254.771,A -85,B 0,C 180,E1 3496.048,E2 3496.048} C_VEL
LIN {X 0,Y 691.282,Z 1277.657,A -85,B 0,C 180,E1 3502.436,E2 3502.436} C_VEL
LIN {X 0,Y 691.186,Z 1286.379,A -85,B 0,C 180,E1 3508.114,E2 3508.114} C_VEL
LIN {X 0,Y 691.233,Z 1283.831,A -85,B 0,C 180,E1 3514.404,E2 3514.404} C_VEL
LIN {X 0,Y 691.229,Z 1269.153,A -85,B 0,C 180,E1 3520.428,E2 3520.428} C_VEL
LIN {X 0,Y 691.738,Z 1241.381,A -85,B 0,C 180,E1 3526.559,E2 3526.559} C_VEL
LIN {X 0,Y 693.178,Z 1200.119,A -85,B 0,C 180,E1 3532.511,E2 3532.511} C_VEL
LIN {X 0,Y 695.751,Z 1145.751,A -85,B 0,C 180,E1 3538.028,E2 3538.028} C_VEL
LIN {X 0,Y 699.298,Z 1080.904,A -85,B 0,C 180,E1 3542.679,E2 3542.679} C_VEL
LIN {X 0,Y 702.795,Z 1010.069,A -85,B 0,C 180,E1 3546.162,E2 3546.162} C_VEL
LIN {X 0,Y 705.326,Z 936.544,A -85,B 0,C 180,E1 3548.391,E2 3548.391} C_VEL
LIN {X 0,Y 704.376,Z 869.975,A -85,B 0,C 180,E1 3549.543,E2 3549.543} C_VEL
LIN {X 0,Y 690.989,Z 844.06,A -85,B 0,C 180,E1 3550.908,E2 3550.908} C_VEL
LIN {X 0,Y 690.78,Z 844.06,A -85,B 0,C 180,E1 3561.279,E2 3561.279} C_VEL
LIN {X 0,Y 690.539,Z 844.06,A -85,B 0,C 180,E1 3568.942,E2 3568.942} C_VEL
LIN {X 0,Y 690.228,Z 844.06,A -85,B 0,C 180,E1 3576.031,E2 3576.031} C_VEL
LIN {X 0,Y 690.788,Z 844.06,A -85,B 0,C 180,E1 3582.776,E2 3582.776} C_VEL
LIN {X 0,Y 690.881,Z 844.06,A -85,B 0,C 180,E1 3590.542,E2 3590.542} C_VEL
LIN {X 0,Y 691.114,Z 844.06,A -85,B 0,C 180,E1 3598.134,E2 3598.134} C_VEL
LIN {X 0,Y 691.072,Z 844.06,A -85,B 0,C 180,E1 3605.69,E2 3605.69} C_VEL
LIN {X 0,Y 690.899,Z 844.06,A -85,B 0,C 180,E1 3613.351,E2 3613.351} C_VEL
LIN {X 0,Y 690.692,Z 844.06,A -85,B 0,C 180,E1 3621.27,E2 3621.27} C_VEL
LIN {X 0,Y 690.515,Z 844.06,A -85,B 0,C 180,E1 3629.829,E2 3629.829} C_VEL
LIN {X 0,Y 690.59,Z 844.06,A -85,B 0,C 180,E1 3637.189,E2 3637.189} C_VEL
LIN {X 0,Y 690.502,Z 844.06,A -85,B 0,C 180,E1 3646.225,E2 3646.225} C_VEL
LIN {X 0,Y 690.068,Z 845.388,A -85,B 0,C 180,E1 3649.228,E2 3649.228} C_VEL
LIN {X 0,Y 705.757,Z 876.382,A -85,B 0,C 180,E1 3650.716,E2 3650.716} C_VEL
LIN {X 0,Y 704.179,Z 957.34,A -85,B 0,C 180,E1 3652.325,E2 3652.325} C_VEL
LIN {X 0,Y 701.201,Z 1032.111,A -85,B 0,C 180,E1 3655.191,E2 3655.191} C_VEL
LIN {X 0,Y 697.616,Z 1101.603,A -85,B 0,C 180,E1 3659.279,E2 3659.279} C_VEL
LIN {X 0,Y 694.443,Z 1163.097,A -85,B 0,C 180,E1 3664.466,E2 3664.466} C_VEL
LIN {X 0,Y 692.319,Z 1210.854,A -85,B 0,C 180,E1 3670.152,E2 3670.152} C_VEL
LIN {X 0,Y 691.352,Z 1243.43,A -85,B 0,C 180,E1 3675.713,E2 3675.713} C_VEL
LIN {X 0,Y 691.104,Z 1265.022,A -85,B 0,C 180,E1 3681.393,E2 3681.393} C_VEL
LIN {X 0,Y 691.025,Z 1275.391,A -85,B 0,C 180,E1 3686.855,E2 3686.855} C_VEL
LIN {X 0,Y 691.058,Z 1275.317,A -85,B 0,C 180,E1 3693.145,E2 3693.145} C_VEL
LIN {X 0,Y 691.072,Z 1264.731,A -85,B 0,C 180,E1 3698.614,E2 3698.614} C_VEL
LIN {X 0,Y 691.407,Z 1241.442,A -85,B 0,C 180,E1 3704.61,E2 3704.61} C_VEL
LIN {X 0,Y 692.53,Z 1205.352,A -85,B 0,C 180,E1 3710.51,E2 3710.51} C_VEL
LIN {X 0,Y 694.775,Z 1155.803,A -85,B 0,C 180,E1 3716.151,E2 3716.151} C_VEL
LIN {X 0,Y 698.008,Z 1094.067,A -85,B 0,C 180,E1 3721.155,E2 3721.155} C_VEL
LIN {X 0,Y 701.641,Z 1024.626,A -85,B 0,C 180,E1 3725.068,E2 3725.068} C_VEL
LIN {X 0,Y 704.54,Z 949.548,A -85,B 0,C 180,E1 3727.793,E2 3727.793} C_VEL
LIN {X 0,Y 703.841,Z 869.858,A -85,B 0,C 180,E1 3729.406,E2 3729.406} C_VEL
LIN {X 0,Y 689.957,Z 844.06,A -85,B 0,C 180,E1 3730.804,E2 3730.804} C_VEL
LIN {X 0,Y 690.25,Z 844.06,A -85,B 0,C 180,E1 3737.88,E2 3737.88} C_VEL
LIN {X 0,Y 690.253,Z 844.06,A -85,B 0,C 180,E1 3745.477,E2 3745.477} C_VEL
LIN {X 0,Y 690.313,Z 844.06,A -85,B 0,C 180,E1 3753.201,E2 3753.201} C_VEL
LIN {X 0,Y 690.492,Z 844.06,A -85,B 0,C 180,E1 3760.069,E2 3760.069} C_VEL
LIN {X 0,Y 691.424,Z 844.06,A -85,B 0,C 180,E1 3767.948,E2 3767.948} C_VEL
LIN {X 0,Y 691.157,Z 844.06,A -85,B 0,C 180,E1 3778.093,E2 3778.093} C_VEL
LIN {X 0,Y 691.066,Z 844.06,A -85,B 0,C 180,E1 3785.649,E2 3785.649} C_VEL
LIN {X 0,Y 690.946,Z 844.06,A -85,B 0,C 180,E1 3793.308,E2 3793.308} C_VEL
LIN {X 0,Y 690.67,Z 844.06,A -85,B 0,C 180,E1 3801.308,E2 3801.308} C_VEL
LIN {X 0,Y 681.966,Z 844.06,A -85,B 0,C 180,E1 3804.18,E2 3804.18} C_VEL
LIN {X 0,Y 682.134,Z 844.06,A -85,B 0,C 180,E1 3811.484,E2 3811.484} C_VEL
LIN {X 0,Y 682.272,Z 844.06,A -85,B 0,C 180,E1 3817.9,E2 3817.9} C_VEL
LIN {X 0,Y 682.432,Z 844.06,A -85,B 0,C 180,E1 3826.229,E2 3826.229} C_VEL
LIN {X 0,Y 682.217,Z 846.102,A -85,B 0,C 180,E1 3828.575,E2 3828.575} C_VEL
LIN {X 0,Y 699.843,Z 879.884,A -85,B 0,C 180,E1 3830.28,E2 3830.28} C_VEL
LIN {X 0,Y 697.775,Z 964.205,A -85,B 0,C 180,E1 3831.87,E2 3831.87} C_VEL
LIN {X 0,Y 694.419,Z 1041.014,A -85,B 0,C 180,E1 3834.79,E2 3834.79} C_VEL
LIN {X 0,Y 690.607,Z 1110.975,A -85,B 0,C 180,E1 3838.932,E2 3838.932} C_VEL
LIN {X 0,Y 687.315,Z 1171.254,A -85,B 0,C 180,E1 3844.044,E2 3844.044} C_VEL
LIN {X 0,Y 685.127,Z 1220.528,A -85,B 0,C 180,E1 3849.934,E2 3849.934} C_VEL
LIN {X 0,Y 683.809,Z 1256.311,A -85,B 0,C 180,E1 3856.207,E2 3856.207} C_VEL
LIN {X 0,Y 683.322,Z 1277.654,A -85,B 0,C 180,E1 3862.348,E2 3862.348} C_VEL
LIN {X 0,Y 683.193,Z 1286.379,A -85,B 0,C 180,E1 3868.092,E2 3868.092} C_VEL
LIN {X 0,Y 683.202,Z 1283.829,A -85,B 0,C 180,E1 3874.456,E2 3874.456} C_VEL
LIN {X 0,Y 683.203,Z 1269.153,A -85,B 0,C 180,E1 3880.552,E2 3880.552} C_VEL
LIN {X 0,Y 683.83,Z 1241.383,A -85,B 0,C 180,E1 3886.756,E2 3886.756} C_VEL
LIN {X 0,Y 685.378,Z 1201.956,A -85,B 0,C 180,E1 3892.548,E2 3892.548} C_VEL
LIN {X 0,Y 688.155,Z 1148.865,A -85,B 0,C 180,E1 3898.078,E2 3898.078} C_VEL
LIN {X 0,Y 692.14,Z 1084.223,A -85,B 0,C 180,E1 3902.85,E2 3902.85} C_VEL
LIN {X 0,Y 695.996,Z 1013.741,A -85,B 0,C 180,E1 3906.411,E2 3906.411} C_VEL
LIN {X 0,Y 698.897,Z 939.534,A -85,B 0,C 180,E1 3908.736,E2 3908.736} C_VEL
LIN {X 0,Y 698.178,Z 873.34,A -85,B 0,C 180,E1 3909.92,E2 3909.92} C_VEL
LIN {X 0,Y 682.963,Z 844.06,A -85,B 0,C 180,E1 3911.457,E2 3911.457} C_VEL
LIN {X 0,Y 682.712,Z 844.06,A -85,B 0,C 180,E1 3920.734,E2 3920.734} C_VEL
LIN {X 0,Y 682.571,Z 844.06,A -85,B 0,C 180,E1 3928.803,E2 3928.803} C_VEL
LIN {X 0,Y 682.351,Z 844.06,A -85,B 0,C 180,E1 3935.736,E2 3935.736} C_VEL
LIN {X 0,Y 682.411,Z 844.06,A -85,B 0,C 180,E1 3943.888,E2 3943.888} C_VEL
LIN {X 0,Y 682.491,Z 844.06,A -85,B 0,C 180,E1 3951.714,E2 3951.714} C_VEL
LIN {X 0,Y 683.123,Z 844.06,A -85,B 0,C 180,E1 3958.112,E2 3958.112} C_VEL
LIN {X 0,Y 683.021,Z 844.06,A -85,B 0,C 180,E1 3965.757,E2 3965.757} C_VEL
LIN {X 0,Y 682.81,Z 844.06,A -85,B 0,C 180,E1 3973.512,E2 3973.512} C_VEL
LIN {X 0,Y 682.564,Z 844.06,A -85,B 0,C 180,E1 3981.536,E2 3981.536} C_VEL
LIN {X 0,Y 682.45,Z 844.06,A -85,B 0,C 180,E1 3990.034,E2 3990.034} C_VEL
LIN {X 0,Y 682.323,Z 844.06,A -85,B 0,C 180,E1 3997.906,E2 3997.906} C_VEL
LIN {X 0,Y 682.479,Z 844.06,A -85,B 0,C 180,E1 4006.284,E2 4006.284} C_VEL
LIN {X 0,Y 682.169,Z 845.661,A -85,B 0,C 180,E1 4008.658,E2 4008.658} C_VEL
LIN {X 0,Y 699.588,Z 878.753,A -85,B 0,C 180,E1 4010.333,E2 4010.333} C_VEL
LIN {X 0,Y 697.708,Z 959.207,A -85,B 0,C 180,E1 4011.973,E2 4011.973} C_VEL
LIN {X 0,Y 694.424,Z 1032.563,A -85,B 0,C 180,E1 4014.824,E2 4014.824} C_VEL
LIN {X 0,Y 690.448,Z 1101.596,A -85,B 0,C 180,E1 4018.925,E2 4018.925} C_VEL
LIN {X 0,Y 686.978,Z 1162.196,A -85,B 0,C 180,E1 4024.079,E2 4024.079} C_VEL
LIN {X 0,Y 684.577,Z 1210.848,A -85,B 0,C 180,E1 4029.918,E2 4029.918} C_VEL
LIN {X 0,Y 683.324,Z 1244.986,A -85,B 0,C 180,E1 4035.87,E2 4035.87} C_VEL
LIN {X 0,Y 682.96,Z 1266.141,A -85,B 0,C 180,E1 4041.701,E2 4041.701} C_VEL
LIN {X 0,Y 683.034,Z 1275.391,A -85,B 0,C 180,E1 4046.818,E2 4046.818} C_VEL
LIN {X 0,Y 683.048,Z 1275.318,A -85,B 0,C 180,E1 4053.182,E2 4053.182} C_VEL
LIN {X 0,Y 682.965,Z 1263.744,A -85,B 0,C 180,E1 4059.046,E2 4059.046} C_VEL
LIN {X 0,Y 683.419,Z 1241.446,A -85,B 0,C 180,E1 4064.785,E2 4064.785} C_VEL
LIN {X 0,Y 684.679,Z 1206.58,A -85,B 0,C 180,E1 4070.587,E2 4070.587} C_VEL
LIN {X 0,Y 687.178,Z 1157.294,A -85,B 0,C 180,E1 4076.314,E2 4076.314} C_VEL
LIN {X 0,Y 690.848,Z 1094.706,A -85,B 0,C 180,E1 4081.469,E2 4081.469} C_VEL
LIN {X 0,Y 694.89,Z 1025.219,A -85,B 0,C 180,E1 4085.43,E2 4085.43} C_VEL
LIN {X 0,Y 698.114,Z 950.504,A -85,B 0,C 180,E1 4088.175,E2 4088.175} C_VEL
LIN {X 0,Y 697.65,Z 873.163,A -85,B 0,C 180,E1 4089.782,E2 4089.782} C_VEL
LIN {X 0,Y 682.005,Z 844.06,A -85,B 0,C 180,E1 4091.325,E2 4091.325} C_VEL
LIN {X 0,Y 682.219,Z 844.06,A -85,B 0,C 180,E1 4098.132,E2 4098.132} C_VEL
LIN {X 0,Y 682.258,Z 844.06,A -85,B 0,C 180,E1 4105.433,E2 4105.433} C_VEL
LIN {X 0,Y 682.375,Z 844.06,A -85,B 0,C 180,E1 4112.864,E2 4112.864} C_VEL
LIN {X 0,Y 682.533,Z 844.06,A -85,B 0,C 180,E1 4119.826,E2 4119.826} C_VEL
LIN {X 0,Y 683.435,Z 844.06,A -85,B 0,C 180,E1 4127.805,E2 4127.805} C_VEL
LIN {X 0,Y 683.165,Z 844.06,A -85,B 0,C 180,E1 4138.071,E2 4138.071} C_VEL
LIN {X 0,Y 683.018,Z 844.06,A -85,B 0,C 180,E1 4145.715,E2 4145.715} C_VEL
LIN {X 0,Y 682.854,Z 844.06,A -85,B 0,C 180,E1 4153.468,E2 4153.468} C_VEL
LIN {X 0,Y 682.581,Z 844.06,A -85,B 0,C 180,E1 4161.491,E2 4161.491} C_VEL
LIN {X 0,Y 681.966,Z 844.06,A -85,B 0,C 180,E1 4164.18,E2 4164.18} C_VEL
LIN {X 0,Y 674.452,Z 844.06,A -85,B 0,C 180,E1 4167.116,E2 4167.116} C_VEL
LIN {X 0,Y 674.343,Z 844.06,A -85,B 0,C 180,E1 4174.98,E2 4174.98} C_VEL
LIN {X 0,Y 674.193,Z 844.06,A -85,B 0,C 180,E1 4183.309,E2 4183.309} C_VEL
LIN {X 0,Y 674.194,Z 845.599,A -85,B 0,C 180,E1 4187.964,E2 4187.964} C_VEL
LIN {X 0,Y 693.689,Z 881.448,A -85,B 0,C 180,E1 4189.877,E2 4189.877} C_VEL
LIN {X 0,Y 691.402,Z 964.806,A -85,B 0,C 180,E1 4191.473,E2 4191.473} C_VEL
LIN {X 0,Y 687.691,Z 1041.387,A -85,B 0,C 180,E1 4194.413,E2 4194.413} C_VEL
LIN {X 0,Y 683.477,Z 1110.977,A -85,B 0,C 180,E1 4198.572,E2 4198.572} C_VEL
LIN {X 0,Y 679.772,Z 1171.738,A -85,B 0,C 180,E1 4203.783,E2 4203.783} C_VEL
LIN {X 0,Y 677.423,Z 1220.526,A -85,B 0,C 180,E1 4209.696,E2 4209.696} C_VEL
LIN {X 0,Y 675.692,Z 1257.795,A -85,B 0,C 180,E1 4216.369,E2 4216.369} C_VEL
LIN {X 0,Y 675.054,Z 1279.164,A -85,B 0,C 180,E1 4222.902,E2 4222.902} C_VEL
LIN {X 0,Y 675.215,Z 1286.379,A -85,B 0,C 180,E1 4228.069,E2 4228.069} C_VEL
LIN {X 0,Y 675.194,Z 1283.827,A -85,B 0,C 180,E1 4234.509,E2 4234.509} C_VEL
LIN {X 0,Y 675.186,Z 1269.152,A -85,B 0,C 180,E1 4240.679,E2 4240.679} C_VEL
LIN {X 0,Y 675.905,Z 1241.6,A -85,B 0,C 180,E1 4246.917,E2 4246.917} C_VEL
LIN {X 0,Y 677.582,Z 1201.471,A -85,B 0,C 180,E1 4252.885,E2 4252.885} C_VEL
LIN {X 0,Y 680.844,Z 1147.994,A -85,B 0,C 180,E1 4258.489,E2 4258.489} C_VEL
LIN {X 0,Y 685.254,Z 1082.197,A -85,B 0,C 180,E1 4263.355,E2 4263.355} C_VEL
LIN {X 0,Y 689.535,Z 1011.821,A -85,B 0,C 180,E1 4266.896,E2 4266.896} C_VEL
LIN {X 0,Y 692.763,Z 937.034,A -85,B 0,C 180,E1 4269.207,E2 4269.207} C_VEL
LIN {X 0,Y 692.226,Z 876.781,A -85,B 0,C 180,E1 4270.288,E2 4270.288} C_VEL
LIN {X 0,Y 674.852,Z 844.06,A -85,B 0,C 180,E1 4272.088,E2 4272.088} C_VEL
LIN {X 0,Y 674.669,Z 844.06,A -85,B 0,C 180,E1 4281.831,E2 4281.831} C_VEL
LIN {X 0,Y 674.449,Z 844.06,A -85,B 0,C 180,E1 4289.962,E2 4289.962} C_VEL
LIN {X 0,Y 674.062,Z 844.06,A -85,B 0,C 180,E1 4296.828,E2 4296.828} C_VEL
LIN {X 0,Y 674.447,Z 844.06,A -85,B 0,C 180,E1 4303.692,E2 4303.692} C_VEL
LIN {X 0,Y 674.529,Z 844.06,A -85,B 0,C 180,E1 4311.615,E2 4311.615} C_VEL
LIN {X 0,Y 675.143,Z 844.06,A -85,B 0,C 180,E1 4318.089,E2 4318.089} C_VEL
LIN {X 0,Y 674.986,Z 844.06,A -85,B 0,C 180,E1 4325.826,E2 4325.826} C_VEL
LIN {X 0,Y 674.726,Z 844.06,A -85,B 0,C 180,E1 4333.677,E2 4333.677} C_VEL
LIN {X 0,Y 674.452,Z 844.06,A -85,B 0,C 180,E1 4341.808,E2 4341.808} C_VEL
LIN {X 0,Y 674.322,Z 844.06,A -85,B 0,C 180,E1 4350.434,E2 4350.434} C_VEL
LIN {X 0,Y 674.209,Z 844.06,A -85,B 0,C 180,E1 4358.253,E2 4358.253} C_VEL
LIN {X 0,Y 674.312,Z 844.06,A -85,B 0,C 180,E1 4367.015,E2 4367.015} C_VEL
LIN {X 0,Y 674.387,Z 846.171,A -85,B 0,C 180,E1 4368.082,E2 4368.082} C_VEL
LIN {X 0,Y 693.482,Z 882.776,A -85,B 0,C 180,E1 4369.967,E2 4369.967} C_VEL
LIN {X 0,Y 691.228,Z 962.513,A -85,B 0,C 180,E1 4371.658,E2 4371.658} C_VEL
LIN {X 0,Y 687.468,Z 1036.666,A -85,B 0,C 180,E1 4374.626,E2 4374.626} C_VEL
LIN {X 0,Y 683.051,Z 1105.733,A -85,B 0,C 180,E1 4378.857,E2 4378.857} C_VEL
LIN {X 0,Y 679.152,Z 1166.198,A -85,B 0,C 180,E1 4384.187,E2 4384.187} C_VEL
LIN {X 0,Y 676.619,Z 1213.113,A -85,B 0,C 180,E1 4390.017,E2 4390.017} C_VEL
LIN {X 0,Y 675.326,Z 1246.52,A -85,B 0,C 180,E1 4396.031,E2 4396.031} C_VEL
LIN {X 0,Y 675.013,Z 1266.14,A -85,B 0,C 180,E1 4401.603,E2 4401.603} C_VEL
LIN {X 0,Y 675.054,Z 1275.39,A -85,B 0,C 180,E1 4406.78,E2 4406.78} C_VEL
LIN {X 0,Y 675.049,Z 1275.318,A -85,B 0,C 180,E1 4413.22,E2 4413.22} C_VEL
LIN {X 0,Y 675.05,Z 1264.96,A -85,B 0,C 180,E1 4418.744,E2 4418.744} C_VEL
LIN {X 0,Y 675.512,Z 1243.006,A -85,B 0,C 180,E1 4424.629,E2 4424.629} C_VEL
LIN {X 0,Y 676.859,Z 1208.111,A -85,B 0,C 180,E1 4430.62,E2 4430.62} C_VEL
LIN {X 0,Y 679.625,Z 1158.318,A -85,B 0,C 180,E1 4436.526,E2 4436.526} C_VEL
LIN {X 0,Y 683.619,Z 1096.495,A -85,B 0,C 180,E1 4441.709,E2 4441.709} C_VEL
LIN {X 0,Y 688.068,Z 1027.146,A -85,B 0,C 180,E1 4445.738,E2 4445.738} C_VEL
LIN {X 0,Y 691.695,Z 951.877,A -85,B 0,C 180,E1 4448.552,E2 4448.552} C_VEL
LIN {X 0,Y 691.527,Z 876.366,A -85,B 0,C 180,E1 4450.164,E2 4450.164} C_VEL
LIN {X 0,Y 674.097,Z 844.06,A -85,B 0,C 180,E1 4451.924,E2 4451.924} C_VEL
LIN {X 0,Y 674.199,Z 844.06,A -85,B 0,C 180,E1 4458.898,E2 4458.898} C_VEL
LIN {X 0,Y 674.212,Z 844.06,A -85,B 0,C 180,E1 4466.521,E2 4466.521} C_VEL
LIN {X 0,Y 674.28,Z 844.06,A -85,B 0,C 180,E1 4473.954,E2 4473.954} C_VEL
LIN {X 0,Y 674.359,Z 844.06,A -85,B 0,C 180,E1 4480.94,E2 4480.94} C_VEL
LIN {X 0,Y 675.414,Z 844.06,A -85,B 0,C 180,E1 4488.972,E2 4488.972} C_VEL
LIN {X 0,Y 675.186,Z 844.06,A -85,B 0,C 180,E1 4498.048,E2 4498.048} C_VEL
LIN {X 0,Y 674.982,Z 844.06,A -85,B 0,C 180,E1 4505.784,E2 4505.784} C_VEL
LIN {X 0,Y 674.768,Z 844.06,A -85,B 0,C 180,E1 4513.633,E2 4513.633} C_VEL
LIN {X 0,Y 674.482,Z 844.06,A -85,B 0,C 180,E1 4521.762,E2 4521.762} C_VEL
LIN {X 0,Y 674.452,Z 844.06,A -85,B 0,C 180,E1 4527.116,E2 4527.116} C_VEL
LIN {X 0,Y 666.339,Z 844.06,A -85,B 0,C 180,E1 4530.085,E2 4530.085} C_VEL
LIN {X 0,Y 666.044,Z 844.06,A -85,B 0,C 180,E1 4538.755,E2 4538.755} C_VEL
LIN {X 0,Y 666.263,Z 845.205,A -85,B 0,C 180,E1 4547.34,E2 4547.34} C_VEL
LIN {X 0,Y 687.574,Z 885.641,A -85,B 0,C 180,E1 4549.502,E2 4549.502} C_VEL
LIN {X 0,Y 684.93,Z 967.693,A -85,B 0,C 180,E1 4551.13,E2 4551.13} C_VEL
LIN {X 0,Y 680.81,Z 1044.213,A -85,B 0,C 180,E1 4554.145,E2 4554.145} C_VEL
LIN {X 0,Y 676.221,Z 1112.955,A -85,B 0,C 180,E1 4558.344,E2 4558.344} C_VEL
LIN {X 0,Y 672.149,Z 1173.661,A -85,B 0,C 180,E1 4563.662,E2 4563.662} C_VEL
LIN {X 0,Y 669.35,Z 1223.209,A -85,B 0,C 180,E1 4569.85,E2 4569.85} C_VEL
LIN {X 0,Y 667.624,Z 1259.152,A -85,B 0,C 180,E1 4576.536,E2 4576.536} C_VEL
LIN {X 0,Y 667.088,Z 1279.164,A -85,B 0,C 180,E1 4582.817,E2 4582.817} C_VEL
LIN {X 0,Y 667.219,Z 1286.38,A -85,B 0,C 180,E1 4588.046,E2 4588.046} C_VEL
LIN {X 0,Y 667.165,Z 1283.824,A -85,B 0,C 180,E1 4594.563,E2 4594.563} C_VEL
LIN {X 0,Y 667.169,Z 1269.151,A -85,B 0,C 180,E1 4600.809,E2 4600.809} C_VEL
LIN {X 0,Y 667.987,Z 1241.867,A -85,B 0,C 180,E1 4607.073,E2 4607.073} C_VEL
LIN {X 0,Y 669.794,Z 1202.819,A -85,B 0,C 180,E1 4612.99,E2 4612.99} C_VEL
LIN {X 0,Y 673.362,Z 1149.314,A -85,B 0,C 180,E1 4618.709,E2 4618.709} C_VEL
LIN {X 0,Y 678.142,Z 1084.489,A -85,B 0,C 180,E1 4623.598,E2 4623.598} C_VEL
LIN {X 0,Y 682.917,Z 1013.164,A -85,B 0,C 180,E1 4627.252,E2 4627.252} C_VEL
LIN {X 0,Y 686.383,Z 939.963,A -85,B 0,C 180,E1 4629.567,E2 4629.567} C_VEL
LIN {X 0,Y 686.03,Z 879.795,A -85,B 0,C 180,E1 4630.687,E2 4630.687} C_VEL
LIN {X 0,Y 666.726,Z 844.06,A -85,B 0,C 180,E1 4632.827,E2 4632.827} C_VEL
LIN {X 0,Y 666.693,Z 844.06,A -85,B 0,C 180,E1 4641.7,E2 4641.7} C_VEL
LIN {X 0,Y 666.458,Z 844.06,A -85,B 0,C 180,E1 4649.217,E2 4649.217} C_VEL
LIN {X 0,Y 666.112,Z 844.06,A -85,B 0,C 180,E1 4656.535,E2 4656.535} C_VEL
LIN {X 0,Y 666.515,Z 844.06,A -85,B 0,C 180,E1 4663.493,E2 4663.493} C_VEL
LIN {X 0,Y 666.47,Z 844.06,A -85,B 0,C 180,E1 4671.822,E2 4671.822} C_VEL
LIN {X 0,Y 667.146,Z 844.06,A -85,B 0,C 180,E1 4678.066,E2 4678.066} C_VEL
LIN {X 0,Y 666.936,Z 844.06,A -85,B 0,C 180,E1 4685.896,E2 4685.896} C_VEL
LIN {X 0,Y 666.646,Z 844.06,A -85,B 0,C 180,E1 4693.846,E2 4693.846} C_VEL
LIN {X 0,Y 666.341,Z 844.06,A -85,B 0,C 180,E1 4702.087,E2 4702.087} C_VEL
LIN {X 0,Y 666.57,Z 844.06,A -85,B 0,C 180,E1 4709.32,E2 4709.32} C_VEL
LIN {X 0,Y 666.229,Z 844.06,A -85,B 0,C 180,E1 4718.25,E2 4718.25} C_VEL
LIN {X 0,Y 666.285,Z 844.06,A -85,B 0,C 180,E1 4727.134,E2 4727.134} C_VEL
LIN {X 0,Y 667.21,Z 847.956,A -85,B 0,C 180,E1 4727.553,E2 4727.553} C_VEL
LIN {X 0,Y 687.369,Z 885.772,A -85,B 0,C 180,E1 4729.583,E2 4729.583} C_VEL
LIN {X 0,Y 684.785,Z 964.457,A -85,B 0,C 180,E1 4731.301,E2 4731.301} C_VEL
LIN {X 0,Y 680.622,Z 1038.665,A -85,B 0,C 180,E1 4734.325,E2 4734.325} C_VEL
LIN {X 0,Y 675.785,Z 1107.183,A -85,B 0,C 180,E1 4738.602,E2 4738.602} C_VEL
LIN {X 0,Y 671.641,Z 1166.194,A -85,B 0,C 180,E1 4743.877,E2 4743.877} C_VEL
LIN {X 0,Y 668.745,Z 1214.391,A -85,B 0,C 180,E1 4749.972,E2 4749.972} C_VEL
LIN {X 0,Y 667.401,Z 1246.651,A -85,B 0,C 180,E1 4755.891,E2 4755.891} C_VEL
LIN {X 0,Y 666.985,Z 1266.876,A -85,B 0,C 180,E1 4761.793,E2 4761.793} C_VEL
LIN {X 0,Y 667.063,Z 1275.39,A -85,B 0,C 180,E1 4766.742,E2 4766.742} C_VEL
LIN {X 0,Y 667.041,Z 1275.318,A -85,B 0,C 180,E1 4773.258,E2 4773.258} C_VEL
LIN {X 0,Y 666.97,Z 1264.06,A -85,B 0,C 180,E1 4779.158,E2 4779.158} C_VEL
LIN {X 0,Y 667.497,Z 1242.482,A -85,B 0,C 180,E1 4784.923,E2 4784.923} C_VEL
LIN {X 0,Y 669.059,Z 1208.295,A -85,B 0,C 180,E1 4790.845,E2 4790.845} C_VEL
LIN {X 0,Y 672.07,Z 1159.293,A -85,B 0,C 180,E1 4796.748,E2 4796.748} C_VEL
LIN {X 0,Y 676.49,Z 1096.812,A -85,B 0,C 180,E1 4802.059,E2 4802.059} C_VEL
LIN {X 0,Y 681.404,Z 1027.156,A -85,B 0,C 180,E1 4806.142,E2 4806.142} C_VEL
LIN {X 0,Y 685.385,Z 952.34,A -85,B 0,C 180,E1 4808.96,E2 4808.96} C_VEL
LIN {X 0,Y 685.523,Z 880.026,A -85,B 0,C 180,E1 4810.54,E2 4810.54} C_VEL
LIN {X 0,Y 666.208,Z 844.06,A -85,B 0,C 180,E1 4812.549,E2 4812.549} C_VEL
LIN {X 0,Y 666.263,Z 844.06,A -85,B 0,C 180,E1 4819.687,E2 4819.687} C_VEL
LIN {X 0,Y 666.312,Z 844.06,A -85,B 0,C 180,E1 4827.628,E2 4827.628} C_VEL
LIN {X 0,Y 666.369,Z 844.06,A -85,B 0,C 180,E1 4835.069,E2 4835.069} C_VEL
LIN {X 0,Y 666.641,Z 844.06,A -85,B 0,C 180,E1 4843.452,E2 4843.452} C_VEL
LIN {X 0,Y 667.152,Z 844.06,A -85,B 0,C 180,E1 4850.159,E2 4850.159} C_VEL
LIN {X 0,Y 667.189,Z 844.06,A -85,B 0,C 180,E1 4858.024,E2 4858.024} C_VEL
LIN {X 0,Y 666.936,Z 844.06,A -85,B 0,C 180,E1 4865.854,E2 4865.854} C_VEL
LIN {X 0,Y 666.689,Z 844.06,A -85,B 0,C 180,E1 4873.801,E2 4873.801} C_VEL
LIN {X 0,Y 666.366,Z 844.06,A -85,B 0,C 180,E1 4882.041,E2 4882.041} C_VEL
LIN {X 0,Y 666.339,Z 844.06,A -85,B 0,C 180,E1 4890.085,E2 4890.085} C_VEL
LIN {X 0,Y 658.028,Z 844.06,A -85,B 0,C 180,E1 4893.06,E2 4893.06} C_VEL
LIN {X 0,Y 657.88,Z 844.06,A -85,B 0,C 180,E1 4899.445,E2 4899.445} C_VEL
LIN {X 0,Y 658.372,Z 844.683,A -85,B 0,C 180,E1 4906.697,E2 4906.697} C_VEL
LIN {X 0,Y 681.517,Z 888.855,A -85,B 0,C 180,E1 4909.11,E2 4909.11} C_VEL
LIN {X 0,Y 678.524,Z 970.138,A -85,B 0,C 180,E1 4910.773,E2 4910.773} C_VEL
LIN {X 0,Y 674.07,Z 1045.622,A -85,B 0,C 180,E1 4913.804,E2 4913.804} C_VEL
LIN {X 0,Y 668.965,Z 1114.964,A -85,B 0,C 180,E1 4918.113,E2 4918.113} C_VEL
LIN {X 0,Y 664.594,Z 1173.972,A -85,B 0,C 180,E1 4923.373,E2 4923.373} C_VEL
LIN {X 0,Y 661.686,Z 1222.857,A -85,B 0,C 180,E1 4929.55,E2 4929.55} C_VEL
LIN {X 0,Y 659.933,Z 1257.797,A -85,B 0,C 180,E1 4936.037,E2 4936.037} C_VEL
LIN {X 0,Y 659.124,Z 1279.164,A -85,B 0,C 180,E1 4942.73,E2 4942.73} C_VEL
LIN {X 0,Y 659.239,Z 1286.38,A -85,B 0,C 180,E1 4948.022,E2 4948.022} C_VEL
LIN {X 0,Y 659.164,Z 1283.821,A -85,B 0,C 180,E1 4954.619,E2 4954.619} C_VEL
LIN {X 0,Y 659.156,Z 1269.151,A -85,B 0,C 180,E1 4960.942,E2 4960.942} C_VEL
LIN {X 0,Y 660.075,Z 1242.663,A -85,B 0,C 180,E1 4967.129,E2 4967.129} C_VEL
LIN {X 0,Y 662.03,Z 1204.169,A -85,B 0,C 180,E1 4973.097,E2 4973.097} C_VEL
LIN {X 0,Y 665.827,Z 1151.692,A -85,B 0,C 180,E1 4978.834,E2 4978.834} C_VEL
LIN {X 0,Y 670.925,Z 1088.232,A -85,B 0,C 180,E1 4983.746,E2 4983.746} C_VEL
LIN {X 0,Y 676.011,Z 1018.602,A -85,B 0,C 180,E1 4987.441,E2 4987.441} C_VEL
LIN {X 0,Y 680.007,Z 943.589,A -85,B 0,C 180,E1 4989.916,E2 4989.916} C_VEL
LIN {X 0,Y 679.929,Z 883.036,A -85,B 0,C 180,E1 4991.086,E2 4991.086} C_VEL
LIN {X 0,Y 658.531,Z 844.06,A -85,B 0,C 180,E1 4993.508,E2 4993.508} C_VEL
LIN {X 0,Y 658.633,Z 844.06,A -85,B 0,C 180,E1 5002.597,E2 5002.597} C_VEL
LIN {X 0,Y 658.414,Z 844.06,A -85,B 0,C 180,E1 5010.33,E2 5010.33} C_VEL
LIN {X 0,Y 658.008,Z 844.06,A -85,B 0,C 180,E1 5017.664,E2 5017.664} C_VEL
LIN {X 0,Y 658.213,Z 844.06,A -85,B 0,C 180,E1 5024.652,E2 5024.652} C_VEL
LIN {X 0,Y 658.564,Z 844.06,A -85,B 0,C 180,E1 5031.41,E2 5031.41} C_VEL
LIN {X 0,Y 659.157,Z 844.06,A -85,B 0,C 180,E1 5038.043,E2 5038.043} C_VEL
LIN {X 0,Y 658.891,Z 844.06,A -85,B 0,C 180,E1 5045.968,E2 5045.968} C_VEL
LIN {X 0,Y 658.599,Z 844.06,A -85,B 0,C 180,E1 5054.018,E2 5054.018} C_VEL
LIN {X 0,Y 658.256,Z 844.06,A -85,B 0,C 180,E1 5062.373,E2 5062.373} C_VEL
LIN {X 0,Y 658.303,Z 844.06,A -85,B 0,C 180,E1 5070.244,E2 5070.244} C_VEL
LIN {X 0,Y 658.297,Z 844.06,A -85,B 0,C 180,E1 5077.666,E2 5077.666} C_VEL
LIN {X 0,Y 658.457,Z 845.159,A -85,B 0,C 180,E1 5086.812,E2 5086.812} C_VEL
LIN {X 0,Y 681.263,Z 890.054,A -85,B 0,C 180,E1 5089.213,E2 5089.213} C_VEL
LIN {X 0,Y 678.311,Z 967.592,A -85,B 0,C 180,E1 5090.978,E2 5090.978} C_VEL
LIN {X 0,Y 673.759,Z 1040.663,A -85,B 0,C 180,E1 5094.022,E2 5094.022} C_VEL
LIN {X 0,Y 668.424,Z 1109.662,A -85,B 0,C 180,E1 5098.422,E2 5098.422} C_VEL
LIN {X 0,Y 663.896,Z 1168.986,A -85,B 0,C 180,E1 5103.864,E2 5103.864} C_VEL
LIN {X 0,Y 660.88,Z 1215.622,A -85,B 0,C 180,E1 5109.918,E2 5109.918} C_VEL
LIN {X 0,Y 659.384,Z 1247.979,A -85,B 0,C 180,E1 5116.025,E2 5116.025} C_VEL
LIN {X 0,Y 658.972,Z 1267.316,A -85,B 0,C 180,E1 5121.878,E2 5121.878} C_VEL
LIN {X 0,Y 659.082,Z 1275.389,A -85,B 0,C 180,E1 5126.702,E2 5126.702} C_VEL
LIN {X 0,Y 659.047,Z 1275.318,A -85,B 0,C 180,E1 5133.298,E2 5133.298} C_VEL
LIN {X 0,Y 658.981,Z 1264.062,A -85,B 0,C 180,E1 5139.27,E2 5139.27} C_VEL
LIN {X 0,Y 659.563,Z 1242.94,A -85,B 0,C 180,E1 5145.008,E2 5145.008} C_VEL
LIN {X 0,Y 661.206,Z 1208.777,A -85,B 0,C 180,E1 5151.034,E2 5151.034} C_VEL
LIN {X 0,Y 664.526,Z 1159.297,A -85,B 0,C 180,E1 5157.076,E2 5157.076} C_VEL
LIN {X 0,Y 669.36,Z 1097.448,A -85,B 0,C 180,E1 5162.394,E2 5162.394} C_VEL
LIN {X 0,Y 674.768,Z 1027.166,A -85,B 0,C 180,E1 5166.554,E2 5166.554} C_VEL
LIN {X 0,Y 679.095,Z 952.912,A -85,B 0,C 180,E1 5169.373,E2 5169.373} C_VEL
LIN {X 0,Y 679.376,Z 883.244,A -85,B 0,C 180,E1 5170.941,E2 5170.941} C_VEL
LIN {X 0,Y 658.398,Z 844.06,A -85,B 0,C 180,E1 5173.218,E2 5173.218} C_VEL
LIN {X 0,Y 658.555,Z 844.06,A -85,B 0,C 180,E1 5182.606,E2 5182.606} C_VEL
LIN {X 0,Y 658.502,Z 844.06,A -85,B 0,C 180,E1 5191.794,E2 5191.794} C_VEL
LIN {X 0,Y 658.396,Z 844.06,A -85,B 0,C 180,E1 5200.46,E2 5200.46} C_VEL
LIN {X 0,Y 659.411,Z 844.06,A -85,B 0,C 180,E1 5208.701,E2 5208.701} C_VEL
LIN {X 0,Y 659.194,Z 844.06,A -85,B 0,C 180,E1 5218,E2 5218} C_VEL
LIN {X 0,Y 658.891,Z 844.06,A -85,B 0,C 180,E1 5225.925,E2 5225.925} C_VEL
LIN {X 0,Y 658.635,Z 844.06,A -85,B 0,C 180,E1 5233.973,E2 5233.973} C_VEL
LIN {X 0,Y 658.301,Z 844.06,A -85,B 0,C 180,E1 5242.325,E2 5242.325} C_VEL
LIN {X 0,Y 658.312,Z 844.06,A -85,B 0,C 180,E1 5250.245,E2 5250.245} C_VEL
LIN {X 0,Y 658.028,Z 844.06,A -85,B 0,C 180,E1 5253.06,E2 5253.06} C_VEL
LIN {X 0,Y 650.252,Z 844.06,A -85,B 0,C 180,E1 5256.1,E2 5256.1} C_VEL
LIN {X 0,Y 650.338,Z 844.805,A -85,B 0,C 180,E1 5266.028,E2 5266.028} C_VEL
LIN {X 0,Y 675.454,Z 893.155,A -85,B 0,C 180,E1 5268.723,E2 5268.723} C_VEL
LIN {X 0,Y 672.092,Z 973.1,A -85,B 0,C 180,E1 5270.425,E2 5270.425} C_VEL
LIN {X 0,Y 667.173,Z 1048.568,A -85,B 0,C 180,E1 5273.532,E2 5273.532} C_VEL
LIN {X 0,Y 661.638,Z 1117.619,A -85,B 0,C 180,E1 5277.935,E2 5277.935} C_VEL
LIN {X 0,Y 656.886,Z 1176.82,A -85,B 0,C 180,E1 5283.362,E2 5283.362} C_VEL
LIN {X 0,Y 653.757,Z 1224.503,A -85,B 0,C 180,E1 5289.555,E2 5289.555} C_VEL
LIN {X 0,Y 651.848,Z 1259.154,A -85,B 0,C 180,E1 5296.204,E2 5296.204} C_VEL
LIN {X 0,Y 651.161,Z 1279.164,A -85,B 0,C 180,E1 5302.64,E2 5302.64} C_VEL
LIN {X 0,Y 651.242,Z 1286.38,A -85,B 0,C 180,E1 5307.998,E2 5307.998} C_VEL
LIN {X 0,Y 651.136,Z 1283.818,A -85,B 0,C 180,E1 5314.676,E2 5314.676} C_VEL
LIN {X 0,Y 651.148,Z 1269.15,A -85,B 0,C 180,E1 5321.078,E2 5321.078} C_VEL
LIN {X 0,Y 652.171,Z 1242.664,A -85,B 0,C 180,E1 5327.343,E2 5327.343} C_VEL
LIN {X 0,Y 654.297,Z 1204.79,A -85,B 0,C 180,E1 5333.303,E2 5333.303} C_VEL
LIN {X 0,Y 658.49,Z 1151.69,A -85,B 0,C 180,E1 5339.187,E2 5339.187} C_VEL
LIN {X 0,Y 664.085,Z 1087.268,A -85,B 0,C 180,E1 5344.21,E2 5344.21} C_VEL
LIN {X 0,Y 669.63,Z 1017.312,A -85,B 0,C 180,E1 5347.922,E2 5347.922} C_VEL
LIN {X 0,Y 673.811,Z 944.434,A -85,B 0,C 180,E1 5350.335,E2 5350.335} C_VEL
LIN {X 0,Y 674.053,Z 886.397,A -85,B 0,C 180,E1 5351.476,E2 5351.476} C_VEL
LIN {X 0,Y 650.33,Z 844.06,A -85,B 0,C 180,E1 5354.126,E2 5354.126} C_VEL
LIN {X 0,Y 650.556,Z 844.06,A -85,B 0,C 180,E1 5361.861,E2 5361.861} C_VEL
LIN {X 0,Y 650.427,Z 844.06,A -85,B 0,C 180,E1 5369.929,E2 5369.929} C_VEL
LIN {X 0,Y 650.004,Z 844.06,A -85,B 0,C 180,E1 5377.374,E2 5377.374} C_VEL
LIN {X 0,Y 650.236,Z 844.06,A -85,B 0,C 180,E1 5384.459,E2 5384.459} C_VEL
LIN {X 0,Y 650.364,Z 844.06,A -85,B 0,C 180,E1 5392.318,E2 5392.318} C_VEL
LIN {X 0,Y 651.159,Z 844.06,A -85,B 0,C 180,E1 5398.019,E2 5398.019} C_VEL
LIN {X 0,Y 650.846,Z 844.06,A -85,B 0,C 180,E1 5406.043,E2 5406.043} C_VEL
LIN {X 0,Y 650.409,Z 844.06,A -85,B 0,C 180,E1 5414.616,E2 5414.616} C_VEL
LIN {X 0,Y 650.141,Z 844.06,A -85,B 0,C 180,E1 5422.871,E2 5422.871} C_VEL
LIN {X 0,Y 650.349,Z 844.06,A -85,B 0,C 180,E1 5430.126,E2 5430.126} C_VEL
LIN {X 0,Y 650.043,Z 844.06,A -85,B 0,C 180,E1 5438.598,E2 5438.598} C_VEL
LIN {X 0,Y 650.579,Z 845.818,A -85,B 0,C 180,E1 5446.168,E2 5446.168} C_VEL
LIN {X 0,Y 675.173,Z 892.357,A -85,B 0,C 180,E1 5448.805,E2 5448.805} C_VEL
LIN {X 0,Y 671.923,Z 969.122,A -85,B 0,C 180,E1 5450.593,E2 5450.593} C_VEL
LIN {X 0,Y 666.928,Z 1042.654,A -85,B 0,C 180,E1 5453.714,E2 5453.714} C_VEL
LIN {X 0,Y 661.195,Z 1110.884,A -85,B 0,C 180,E1 5458.14,E2 5458.14} C_VEL
LIN {X 0,Y 656.204,Z 1171.034,A -85,B 0,C 180,E1 5463.769,E2 5463.769} C_VEL
LIN {X 0,Y 653.049,Z 1216.398,A -85,B 0,C 180,E1 5469.792,E2 5469.792} C_VEL
LIN {X 0,Y 651.457,Z 1247.977,A -85,B 0,C 180,E1 5475.852,E2 5475.852} C_VEL
LIN {X 0,Y 650.992,Z 1267.527,A -85,B 0,C 180,E1 5481.871,E2 5481.871} C_VEL
LIN {X 0,Y 651.09,Z 1275.388,A -85,B 0,C 180,E1 5486.662,E2 5486.662} C_VEL
LIN {X 0,Y 651.256,Z 1276.345,A -85,B 0,C 180,E1 5492.002,E2 5492.002} C_VEL
LIN {X 0,Y 651.332,Z 1267.595,A -85,B 0,C 180,E1 5498.006,E2 5498.006} C_VEL
LIN {X 0,Y 651.672,Z 1246.047,A -85,B 0,C 180,E1 5504.501,E2 5504.501} C_VEL
LIN {X 0,Y 653.353,Z 1211.381,A -85,B 0,C 180,E1 5510.914,E2 5510.914} C_VEL
LIN {X 0,Y 656.882,Z 1162.696,A -85,B 0,C 180,E1 5517.058,E2 5517.058} C_VEL
LIN {X 0,Y 662.004,Z 1101.561,A -85,B 0,C 180,E1 5522.481,E2 5522.481} C_VEL
LIN {X 0,Y 667.774,Z 1032.796,A -85,B 0,C 180,E1 5526.699,E2 5526.699} C_VEL
LIN {X 0,Y 672.562,Z 958.251,A -85,B 0,C 180,E1 5529.66,E2 5529.66} C_VEL
LIN {X 0,Y 673.509,Z 886.798,A -85,B 0,C 180,E1 5531.321,E2 5531.321} C_VEL
LIN {X 0,Y 650.432,Z 844.06,A -85,B 0,C 180,E1 5533.901,E2 5533.901} C_VEL
LIN {X 0,Y 650.461,Z 844.06,A -85,B 0,C 180,E1 5543.48,E2 5543.48} C_VEL
LIN {X 0,Y 650.479,Z 844.06,A -85,B 0,C 180,E1 5551.414,E2 5551.414} C_VEL
LIN {X 0,Y 650.408,Z 844.06,A -85,B 0,C 180,E1 5560.21,E2 5560.21} C_VEL
LIN {X 0,Y 651.399,Z 844.06,A -85,B 0,C 180,E1 5568.561,E2 5568.561} C_VEL
LIN {X 0,Y 651.196,Z 844.06,A -85,B 0,C 180,E1 5577.976,E2 5577.976} C_VEL
LIN {X 0,Y 650.849,Z 844.06,A -85,B 0,C 180,E1 5585.999,E2 5585.999} C_VEL
LIN {X 0,Y 650.407,Z 844.06,A -85,B 0,C 180,E1 5594.615,E2 5594.615} C_VEL
LIN {X 0,Y 650.203,Z 844.06,A -85,B 0,C 180,E1 5602.618,E2 5602.618} C_VEL
LIN {X 0,Y 650.353,Z 844.06,A -85,B 0,C 180,E1 5610.075,E2 5610.075} C_VEL
LIN {X 0,Y 650.252,Z 844.06,A -85,B 0,C 180,E1 5616.1,E2 5616.1} C_VEL
LIN {X 0,Y 641.867,Z 844.06,A -85,B 0,C 180,E1 5619.164,E2 5619.164} C_VEL
LIN {X 0,Y 642.43,Z 845.426,A -85,B 0,C 180,E1 5625.353,E2 5625.353} C_VEL
LIN {X 0,Y 669.394,Z 896.808,A -85,B 0,C 180,E1 5628.324,E2 5628.324} C_VEL
LIN {X 0,Y 665.599,Z 976.335,A -85,B 0,C 180,E1 5630.084,E2 5630.084} C_VEL
LIN {X 0,Y 660.179,Z 1052.397,A -85,B 0,C 180,E1 5633.313,E2 5633.313} C_VEL
LIN {X 0,Y 654.217,Z 1121.086,A -85,B 0,C 180,E1 5637.822,E2 5637.822} C_VEL
LIN {X 0,Y 649.054,Z 1180.547,A -85,B 0,C 180,E1 5643.447,E2 5643.447} C_VEL
LIN {X 0,Y 645.595,Z 1227.687,A -85,B 0,C 180,E1 5649.804,E2 5649.804} C_VEL
LIN {X 0,Y 643.766,Z 1260.51,A -85,B 0,C 180,E1 5656.375,E2 5656.375} C_VEL
LIN {X 0,Y 642.983,Z 1280.523,A -85,B 0,C 180,E1 5663.227,E2 5663.227} C_VEL
LIN {X 0,Y 643.252,Z 1286.38,A -85,B 0,C 180,E1 5667.973,E2 5667.973} C_VEL
LIN {X 0,Y 643.109,Z 1283.815,A -85,B 0,C 180,E1 5674.734,E2 5674.734} C_VEL
LIN {X 0,Y 643.15,Z 1269.15,A -85,B 0,C 180,E1 5681.217,E2 5681.217} C_VEL
LIN {X 0,Y 644.245,Z 1243.732,A -85,B 0,C 180,E1 5687.35,E2 5687.35} C_VEL
LIN {X 0,Y 646.528,Z 1206.439,A -85,B 0,C 180,E1 5693.373,E2 5693.373} C_VEL
LIN {X 0,Y 650.979,Z 1153.729,A -85,B 0,C 180,E1 5699.353,E2 5699.353} C_VEL
LIN {X 0,Y 656.972,Z 1089.93,A -85,B 0,C 180,E1 5704.44,E2 5704.44} C_VEL
LIN {X 0,Y 662.979,Z 1019.804,A -85,B 0,C 180,E1 5708.249,E2 5708.249} C_VEL
LIN {X 0,Y 667.582,Z 946.229,A -85,B 0,C 180,E1 5710.741,E2 5710.741} C_VEL
LIN {X 0,Y 668.048,Z 889.694,A -85,B 0,C 180,E1 5711.886,E2 5711.886} C_VEL
LIN {X 0,Y 642.155,Z 844.06,A -85,B 0,C 180,E1 5714.809,E2 5714.809} C_VEL
LIN {X 0,Y 642.547,Z 844.06,A -85,B 0,C 180,E1 5723.011,E2 5723.011} C_VEL
LIN {X 0,Y 642.423,Z 844.06,A -85,B 0,C 180,E1 5731.072,E2 5731.072} C_VEL
LIN {X 0,Y 642.369,Z 844.06,A -85,B 0,C 180,E1 5739.998,E2 5739.998} C_VEL
LIN {X 0,Y 642.69,Z 844.06,A -85,B 0,C 180,E1 5748.448,E2 5748.448} C_VEL
LIN {X 0,Y 643.184,Z 844.06,A -85,B 0,C 180,E1 5757.994,E2 5757.994} C_VEL
LIN {X 0,Y 642.826,Z 844.06,A -85,B 0,C 180,E1 5766.118,E2 5766.118} C_VEL
LIN {X 0,Y 642.5,Z 844.06,A -85,B 0,C 180,E1 5774.377,E2 5774.377} C_VEL
LIN {X 0,Y 642.118,Z 844.06,A -85,B 0,C 180,E1 5782.967,E2 5782.967} C_VEL
LIN {X 0,Y 642.246,Z 844.06,A -85,B 0,C 180,E1 5790.546,E2 5790.546} C_VEL
LIN {X 0,Y 641.989,Z 844.06,A -85,B 0,C 180,E1 5798.798,E2 5798.798} C_VEL
LIN {X 0,Y 642.493,Z 845.502,A -85,B 0,C 180,E1 5805.468,E2 5805.468} C_VEL
LIN {X 0,Y 669.1,Z 895.559,A -85,B 0,C 180,E1 5808.403,E2 5808.403} C_VEL
LIN {X 0,Y 665.517,Z 971.287,A -85,B 0,C 180,E1 5810.221,E2 5810.221} C_VEL
LIN {X 0,Y 660.129,Z 1044.525,A -85,B 0,C 180,E1 5813.393,E2 5813.393} C_VEL
LIN {X 0,Y 653.911,Z 1112.767,A -85,B 0,C 180,E1 5817.903,E2 5817.903} C_VEL
LIN {X 0,Y 648.562,Z 1172.629,A -85,B 0,C 180,E1 5823.623,E2 5823.623} C_VEL
LIN {X 0,Y 645.184,Z 1217.492,A -85,B 0,C 180,E1 5829.714,E2 5829.714} C_VEL
LIN {X 0,Y 643.453,Z 1249.332,A -85,B 0,C 180,E1 5836.02,E2 5836.02} C_VEL
LIN {X 0,Y 642.934,Z 1268.427,A -85,B 0,C 180,E1 5842.162,E2 5842.162} C_VEL
LIN {X 0,Y 642.734,Z 1276.414,A -85,B 0,C 180,E1 5847.972,E2 5847.972} C_VEL
LIN {X 0,Y 643.047,Z 1275.319,A -85,B 0,C 180,E1 5853.38,E2 5853.38} C_VEL
LIN {X 0,Y 642.991,Z 1264.064,A -85,B 0,C 180,E1 5859.503,E2 5859.503} C_VEL
LIN {X 0,Y 643.645,Z 1242.963,A -85,B 0,C 180,E1 5865.385,E2 5865.385} C_VEL
LIN {X 0,Y 645.542,Z 1210.218,A -85,B 0,C 180,E1 5871.354,E2 5871.354} C_VEL
LIN {X 0,Y 649.428,Z 1161.377,A -85,B 0,C 180,E1 5877.536,E2 5877.536} C_VEL
LIN {X 0,Y 655.046,Z 1100.411,A -85,B 0,C 180,E1 5882.961,E2 5882.961} C_VEL
LIN {X 0,Y 661.345,Z 1030.649,A -85,B 0,C 180,E1 5887.234,E2 5887.234} C_VEL
LIN {X 0,Y 666.449,Z 956.109,A -85,B 0,C 180,E1 5890.167,E2 5890.167} C_VEL
LIN {X 0,Y 667.582,Z 890.412,A -85,B 0,C 180,E1 5891.709,E2 5891.709} C_VEL
LIN {X 0,Y 642.477,Z 844.06,A -85,B 0,C 180,E1 5894.611,E2 5894.611} C_VEL
LIN {X 0,Y 642.376,Z 844.06,A -85,B 0,C 180,E1 5902.945,E2 5902.945} C_VEL
LIN {X 0,Y 642.495,Z 844.06,A -85,B 0,C 180,E1 5911.026,E2 5911.026} C_VEL
LIN {X 0,Y 642.421,Z 844.06,A -85,B 0,C 180,E1 5919.953,E2 5919.953} C_VEL
LIN {X 0,Y 643.375,Z 844.06,A -85,B 0,C 180,E1 5928.416,E2 5928.416} C_VEL
LIN {X 0,Y 643.218,Z 844.06,A -85,B 0,C 180,E1 5937.951,E2 5937.951} C_VEL
LIN {X 0,Y 642.829,Z 844.06,A -85,B 0,C 180,E1 5946.074,E2 5946.074} C_VEL
LIN {X 0,Y 642.518,Z 844.06,A -85,B 0,C 180,E1 5954.331,E2 5954.331} C_VEL
LIN {X 0,Y 642.15,Z 844.06,A -85,B 0,C 180,E1 5962.918,E2 5962.918} C_VEL
LIN {X 0,Y 642.263,Z 844.06,A -85,B 0,C 180,E1 5970.494,E2 5970.494} C_VEL
LIN {X 0,Y 641.867,Z 844.06,A -85,B 0,C 180,E1 5979.164,E2 5979.164} C_VEL
LIN {X 0,Y 633.791,Z 844.06,A -85,B 0,C 180,E1 5982.276,E2 5982.276} C_VEL
LIN {X 0,Y 634.49,Z 845.934,A -85,B 0,C 180,E1 5984.65,E2 5984.65} C_VEL
LIN {X 0,Y 663.367,Z 899.494,A -85,B 0,C 180,E1 5987.905,E2 5987.905} C_VEL
LIN {X 0,Y 659.276,Z 978.256,A -85,B 0,C 180,E1 5989.697,E2 5989.697} C_VEL
LIN {X 0,Y 653.456,Z 1053.74,A -85,B 0,C 180,E1 5992.955,E2 5992.955} C_VEL
LIN {X 0,Y 646.998,Z 1122.471,A -85,B 0,C 180,E1 5997.539,E2 5997.539} C_VEL
LIN {X 0,Y 641.581,Z 1180.637,A -85,B 0,C 180,E1 6003.124,E2 6003.124} C_VEL
LIN {X 0,Y 637.786,Z 1228.306,A -85,B 0,C 180,E1 6009.65,E2 6009.65} C_VEL
LIN {X 0,Y 635.675,Z 1261.86,A -85,B 0,C 180,E1 6016.549,E2 6016.549} C_VEL
LIN {X 0,Y 635.017,Z 1280.523,A -85,B 0,C 180,E1 6023.142,E2 6023.142} C_VEL
LIN {X 0,Y 635.254,Z 1286.38,A -85,B 0,C 180,E1 6027.948,E2 6027.948} C_VEL
LIN {X 0,Y 635.084,Z 1283.812,A -85,B 0,C 180,E1 6034.794,E2 6034.794} C_VEL
LIN {X 0,Y 635.157,Z 1269.149,A -85,B 0,C 180,E1 6041.36,E2 6041.36} C_VEL
LIN {X 0,Y 636.325,Z 1243.733,A -85,B 0,C 180,E1 6047.573,E2 6047.573} C_VEL
LIN {X 0,Y 638.824,Z 1206.205,A -85,B 0,C 180,E1 6053.704,E2 6053.704} C_VEL
LIN {X 0,Y 643.692,Z 1154.008,A -85,B 0,C 180,E1 6059.69,E2 6059.69} C_VEL
LIN {X 0,Y 650.121,Z 1089.928,A -85,B 0,C 180,E1 6064.856,E2 6064.856} C_VEL
LIN {X 0,Y 656.529,Z 1020.385,A -85,B 0,C 180,E1 6068.665,E2 6068.665} C_VEL
LIN {X 0,Y 661.483,Z 946.29,A -85,B 0,C 180,E1 6071.196,E2 6071.196} C_VEL
LIN {X 0,Y 661.856,Z 892.463,A -85,B 0,C 180,E1 6072.329,E2 6072.329} C_VEL
LIN {X 0,Y 634.06,Z 844.06,A -85,B 0,C 180,E1 6075.587,E2 6075.587} C_VEL
LIN {X 0,Y 634.573,Z 844.06,A -85,B 0,C 180,E1 6084.175,E2 6084.175} C_VEL
LIN {X 0,Y 634.482,Z 844.06,A -85,B 0,C 180,E1 6092.235,E2 6092.235} C_VEL
LIN {X 0,Y 634.574,Z 844.06,A -85,B 0,C 180,E1 6101.195,E2 6101.195} C_VEL
LIN {X 0,Y 634.596,Z 844.06,A -85,B 0,C 180,E1 6111.083,E2 6111.083} C_VEL
LIN {X 0,Y 635.184,Z 844.06,A -85,B 0,C 180,E1 6117.969,E2 6117.969} C_VEL
LIN {X 0,Y 634.783,Z 844.06,A -85,B 0,C 180,E1 6126.196,E2 6126.196} C_VEL
LIN {X 0,Y 634.449,Z 844.06,A -85,B 0,C 180,E1 6134.564,E2 6134.564} C_VEL
LIN {X 0,Y 634.118,Z 844.06,A -85,B 0,C 180,E1 6142.964,E2 6142.964} C_VEL
LIN {X 0,Y 634.132,Z 844.06,A -85,B 0,C 180,E1 6150.979,E2 6150.979} C_VEL
LIN {X 0,Y 633.903,Z 844.06,A -85,B 0,C 180,E1 6159.388,E2 6159.388} C_VEL
LIN {X 0,Y 634.441,Z 845.619,A -85,B 0,C 180,E1 6164.75,E2 6164.75} C_VEL
LIN {X 0,Y 663.074,Z 899.182,A -85,B 0,C 180,E1 6168.002,E2 6168.002} C_VEL
LIN {X 0,Y 659.111,Z 974.358,A -85,B 0,C 180,E1 6169.874,E2 6169.874} C_VEL
LIN {X 0,Y 653.24,Z 1047.476,A -85,B 0,C 180,E1 6173.123,E2 6173.123} C_VEL
LIN {X 0,Y 646.509,Z 1116.15,A -85,B 0,C 180,E1 6177.784,E2 6177.784} C_VEL
LIN {X 0,Y 640.93,Z 1174.225,A -85,B 0,C 180,E1 6183.474,E2 6183.474} C_VEL
LIN {X 0,Y 637.248,Z 1219.66,A -85,B 0,C 180,E1 6189.814,E2 6189.814} C_VEL
LIN {X 0,Y 635.514,Z 1249.331,A -85,B 0,C 180,E1 6195.842,E2 6195.842} C_VEL
LIN {X 0,Y 635.043,Z 1267.738,A -85,B 0,C 180,E1 6201.762,E2 6201.762} C_VEL
LIN {X 0,Y 634.738,Z 1276.414,A -85,B 0,C 180,E1 6207.946,E2 6207.946} C_VEL
LIN {X 0,Y 635.04,Z 1275.319,A -85,B 0,C 180,E1 6213.423,E2 6213.423} C_VEL
LIN {X 0,Y 635.004,Z 1264.065,A -85,B 0,C 180,E1 6219.624,E2 6219.624} C_VEL
LIN {X 0,Y 635.739,Z 1242.829,A -85,B 0,C 180,E1 6225.612,E2 6225.612} C_VEL
LIN {X 0,Y 637.855,Z 1208.692,A -85,B 0,C 180,E1 6231.857,E2 6231.857} C_VEL
LIN {X 0,Y 642.071,Z 1160.299,A -85,B 0,C 180,E1 6237.997,E2 6237.997} C_VEL
LIN {X 0,Y 648.286,Z 1098.313,A -85,B 0,C 180,E1 6243.517,E2 6243.517} C_VEL
LIN {X 0,Y 654.969,Z 1028.923,A -85,B 0,C 180,E1 6247.754,E2 6247.754} C_VEL
LIN {X 0,Y 660.432,Z 954.759,A -85,B 0,C 180,E1 6250.654,E2 6250.654} C_VEL
LIN {X 0,Y 661.383,Z 893.422,A -85,B 0,C 180,E1 6252.138,E2 6252.138} C_VEL
LIN {X 0,Y 634.419,Z 844.06,A -85,B 0,C 180,E1 6255.354,E2 6255.354} C_VEL
LIN {X 0,Y 634.267,Z 844.06,A -85,B 0,C 180,E1 6264.1,E2 6264.1} C_VEL
LIN {X 0,Y 634.345,Z 844.06,A -85,B 0,C 180,E1 6272.178,E2 6272.178} C_VEL
LIN {X 0,Y 634.448,Z 844.06,A -85,B 0,C 180,E1 6279.69,E2 6279.69} C_VEL
LIN {X 0,Y 635.357,Z 844.06,A -85,B 0,C 180,E1 6288.268,E2 6288.268} C_VEL
LIN {X 0,Y 635.219,Z 844.06,A -85,B 0,C 180,E1 6297.925,E2 6297.925} C_VEL
LIN {X 0,Y 634.789,Z 844.06,A -85,B 0,C 180,E1 6306.151,E2 6306.151} C_VEL
LIN {X 0,Y 634.455,Z 844.06,A -85,B 0,C 180,E1 6314.517,E2 6314.517} C_VEL
LIN {X 0,Y 634.139,Z 844.06,A -85,B 0,C 180,E1 6322.968,E2 6322.968} C_VEL
LIN {X 0,Y 634.149,Z 844.06,A -85,B 0,C 180,E1 6330.927,E2 6330.927} C_VEL
LIN {X 0,Y 633.872,Z 844.06,A -85,B 0,C 180,E1 6339.333,E2 6339.333} C_VEL
LIN {X 0,Y 633.791,Z 844.06,A -85,B 0,C 180,E1 6342.276,E2 6342.276} C_VEL
LIN {X 0,Y 626.101,Z 844.06,A -85,B 0,C 180,E1 6343.663,E2 6343.663} C_VEL
LIN {X 0,Y 657.393,Z 901.518,A -85,B 0,C 180,E1 6347.469,E2 6347.469} C_VEL
LIN {X 0,Y 652.947,Z 980.656,A -85,B 0,C 180,E1 6349.318,E2 6349.318} C_VEL
LIN {X 0,Y 646.62,Z 1056.34,A -85,B 0,C 180,E1 6352.658,E2 6352.658} C_VEL
LIN {X 0,Y 639.769,Z 1124.317,A -85,B 0,C 180,E1 6357.288,E2 6357.288} C_VEL
LIN {X 0,Y 633.942,Z 1182.238,A -85,B 0,C 180,E1 6362.966,E2 6362.966} C_VEL
LIN {X 0,Y 629.92,Z 1229.391,A -85,B 0,C 180,E1 6369.568,E2 6369.568} C_VEL
LIN {X 0,Y 627.806,Z 1261.859,A -85,B 0,C 180,E1 6376.378,E2 6376.378} C_VEL
LIN {X 0,Y 627.054,Z 1280.523,A -85,B 0,C 180,E1 6383.054,E2 6383.054} C_VEL
LIN {X 0,Y 626.72,Z 1286.838,A -85,B 0,C 180,E1 6389.307,E2 6389.307} C_VEL
LIN {X 0,Y 626.891,Z 1282.883,A -85,B 0,C 180,E1 6395.553,E2 6395.553} C_VEL
LIN {X 0,Y 627.189,Z 1268,A -85,B 0,C 180,E1 6401.86,E2 6401.86} C_VEL
LIN {X 0,Y 628.468,Z 1243.336,A -85,B 0,C 180,E1 6407.882,E2 6407.882} C_VEL
LIN {X 0,Y 631.354,Z 1204.959,A -85,B 0,C 180,E1 6414.179,E2 6414.179} C_VEL
LIN {X 0,Y 636.557,Z 1152.256,A -85,B 0,C 180,E1 6420.237,E2 6420.237} C_VEL
LIN {X 0,Y 643.461,Z 1088.485,A -85,B 0,C 180,E1 6425.377,E2 6425.377} C_VEL
LIN {X 0,Y 650.156,Z 1020.169,A -85,B 0,C 180,E1 6429.127,E2 6429.127} C_VEL
LIN {X 0,Y 655.453,Z 946.269,A -85,B 0,C 180,E1 6431.659,E2 6431.659} C_VEL
LIN {X 0,Y 656.078,Z 895.964,A -85,B 0,C 180,E1 6432.733,E2 6432.733} C_VEL
LIN {X 0,Y 626.016,Z 844.06,A -85,B 0,C 180,E1 6436.35,E2 6436.35} C_VEL
LIN {X 0,Y 626.587,Z 844.06,A -85,B 0,C 180,E1 6444.175,E2 6444.175} C_VEL
LIN {X 0,Y 626.471,Z 844.06,A -85,B 0,C 180,E1 6453.411,E2 6453.411} C_VEL
LIN {X 0,Y 626.458,Z 844.06,A -85,B 0,C 180,E1 6462.983,E2 6462.983} C_VEL
LIN {X 0,Y 626.601,Z 844.06,A -85,B 0,C 180,E1 6470.969,E2 6470.969} C_VEL
LIN {X 0,Y 627.204,Z 844.06,A -85,B 0,C 180,E1 6477.943,E2 6477.943} C_VEL
LIN {X 0,Y 626.756,Z 844.06,A -85,B 0,C 180,E1 6486.276,E2 6486.276} C_VEL
LIN {X 0,Y 626.383,Z 844.06,A -85,B 0,C 180,E1 6494.755,E2 6494.755} C_VEL
LIN {X 0,Y 626.28,Z 844.06,A -85,B 0,C 180,E1 6502.077,E2 6502.077} C_VEL
LIN {X 0,Y 626.142,Z 844.06,A -85,B 0,C 180,E1 6510.704,E2 6510.704} C_VEL
LIN {X 0,Y 626.061,Z 844.06,A -85,B 0,C 180,E1 6518.192,E2 6518.192} C_VEL
LIN {X 0,Y 626.423,Z 845.913,A -85,B 0,C 180,E1 6524.009,E2 6524.009} C_VEL
LIN {X 0,Y 657.072,Z 902.308,A -85,B 0,C 180,E1 6527.586,E2 6527.586} C_VEL
LIN {X 0,Y 652.694,Z 977.411,A -85,B 0,C 180,E1 6529.518,E2 6529.518} C_VEL
LIN {X 0,Y 646.479,Z 1049.172,A -85,B 0,C 180,E1 6532.778,E2 6532.778} C_VEL
LIN {X 0,Y 639.378,Z 1116.643,A -85,B 0,C 180,E1 6537.424,E2 6537.424} C_VEL
LIN {X 0,Y 633.452,Z 1174.295,A -85,B 0,C 180,E1 6543.145,E2 6543.145} C_VEL
LIN {X 0,Y 629.442,Z 1219.655,A -85,B 0,C 180,E1 6549.552,E2 6549.552} C_VEL
LIN {X 0,Y 627.593,Z 1249.33,A -85,B 0,C 180,E1 6555.66,E2 6555.66} C_VEL
LIN {X 0,Y 627.084,Z 1267.734,A -85,B 0,C 180,E1 6561.657,E2 6561.657} C_VEL
LIN {X 0,Y 626.742,Z 1276.414,A -85,B 0,C 180,E1 6567.92,E2 6567.92} C_VEL
LIN {X 0,Y 627.034,Z 1275.319,A -85,B 0,C 180,E1 6573.467,E2 6573.467} C_VEL
LIN {X 0,Y 627.077,Z 1265.919,A -85,B 0,C 180,E1 6579.044,E2 6579.044} C_VEL
LIN {X 0,Y 627.783,Z 1246.408,A -85,B 0,C 180,E1 6584.982,E2 6584.982} C_VEL
LIN {X 0,Y 629.864,Z 1212.545,A -85,B 0,C 180,E1 6591.542,E2 6591.542} C_VEL
LIN {X 0,Y 634.245,Z 1165.42,A -85,B 0,C 180,E1 6597.792,E2 6597.792} C_VEL
LIN {X 0,Y 640.678,Z 1104.847,A -85,B 0,C 180,E1 6603.44,E2 6603.44} C_VEL
LIN {X 0,Y 647.783,Z 1036.679,A -85,B 0,C 180,E1 6607.813,E2 6607.813} C_VEL
LIN {X 0,Y 653.726,Z 962.781,A -85,B 0,C 180,E1 6610.886,E2 6610.886} C_VEL
LIN {X 0,Y 655.458,Z 896.788,A -85,B 0,C 180,E1 6612.55,E2 6612.55} C_VEL
LIN {X 0,Y 626.396,Z 844.06,A -85,B 0,C 180,E1 6616.144,E2 6616.144} C_VEL
LIN {X 0,Y 626.169,Z 844.06,A -85,B 0,C 180,E1 6625.269,E2 6625.269} C_VEL
LIN {X 0,Y 626.234,Z 844.06,A -85,B 0,C 180,E1 6633.349,E2 6633.349} C_VEL
LIN {X 0,Y 626.344,Z 844.06,A -85,B 0,C 180,E1 6640.891,E2 6640.891} C_VEL
LIN {X 0,Y 627.357,Z 844.06,A -85,B 0,C 180,E1 6648.244,E2 6648.244} C_VEL
LIN {X 0,Y 627.236,Z 844.06,A -85,B 0,C 180,E1 6657.898,E2 6657.898} C_VEL
LIN {X 0,Y 626.76,Z 844.06,A -85,B 0,C 180,E1 6666.23,E2 6666.23} C_VEL
LIN {X 0,Y 626.392,Z 844.06,A -85,B 0,C 180,E1 6674.709,E2 6674.709} C_VEL
LIN {X 0,Y 626.308,Z 844.06,A -85,B 0,C 180,E1 6682.027,E2 6682.027} C_VEL
LIN {X 0,Y 626.174,Z 844.06,A -85,B 0,C 180,E1 6690.708,E2 6690.708} C_VEL
